		// Prepare Data for writing
		// Repetition ID
		IF (SIf.Cur.dwoJob = RFID_Data.cRFID_AllData) OR (SIf.Cur.dwoJob = RFID_Data.cRFID_RepetionID) THEN
			uinDataAdress := DWORD_TO_UINT(RFID_Data.cRFID_RepetionID);
			uinDataAdress := uinDataAdress MOD 16#100;							// Maximum 255 data
			SIf.Cur.abytData[uinDataAdress] := SIf.Cur.stData.usiRepetitionID;
		END_IF
		// Tray Info
		IF (SIf.Cur.dwoJob = RFID_Data.cRFID_AllData) OR (SIf.Cur.dwoJob = RFID_Data.cRFID_TrayInfo) THEN
			uinDataAdress := DWORD_TO_UINT(RFID_Data.cRFID_TrayInfo);
			uinDataAdress := uinDataAdress MOD 16#100;							// Maximum 255 data
			SIf.Cur.abytData[uinDataAdress].0 := SIf.Cur.stData.bolWorkstation2;
			SIf.Cur.abytData[uinDataAdress].6 := SIf.Cur.stData.bolDeleteFileAfterPrint;
			SIf.Cur.abytData[uinDataAdress].7 := SIf.Cur.stData.bolPrintOk;
		END_IF
		// Height of tray
		IF (SIf.Cur.dwoJob = RFID_Data.cRFID_AllData) OR (SIf.Cur.dwoJob = RFID_Data.cRFID_HeighOfTray) THEN
			uinDataAdress := DWORD_TO_UINT(RFID_Data.cRFID_HeighOfTray);
			uinDataAdress := uinDataAdress MOD 16#100;							// Maximum 255 data
			SIf.Cur.abytData[uinDataAdress] := SHL(SIf.Cur.stData.usiHeightOffset,1);
			SIf.Cur.abytData[uinDataAdress].0 := SIf.Cur.stData.bolHeightUseMeasure;
			SIf.Cur.abytData[uinDataAdress].4 := SIf.Cur.stData.bolHeightOffsetSignMinus;
		END_IF
		// Pretreatment
		IF (SIf.Cur.dwoJob = RFID_Data.cRFID_AllData) OR (SIf.Cur.dwoJob = RFID_Data.cRFID_Pretreatment) THEN
			uinDataAdress := DWORD_TO_UINT(RFID_Data.cRFID_Pretreatment);
			uinDataAdress := uinDataAdress MOD 16#100;							// Maximum 255 data
			SIf.Cur.abytData[uinDataAdress] := SHL(SIf.Cur.stData.usiPlasmaLevel,2);
			SIf.Cur.abytData[uinDataAdress].1 := SIf.Cur.stData.bolIonizer;
			SIf.Cur.abytData[uinDataAdress].4 := SIf.Cur.stData.bolPrintPass;
			SIf.Cur.abytData[uinDataAdress].5 := SIf.Cur.stData.bolNozzleCheck;
			SIf.Cur.abytData[uinDataAdress].6 := SIf.Cur.stData.bolAligneCheck;
		END_IF
		// UV-curing
		IF (SIf.Cur.dwoJob = RFID_Data.cRFID_AllData) OR (SIf.Cur.dwoJob = RFID_Data.cRFID_UVcuring) THEN
			uinDataAdress := DWORD_TO_UINT(RFID_Data.cRFID_UVcuring);
			uinDataAdress := uinDataAdress MOD 16#100;							// Maximum 255 data
			SIf.Cur.abytData[uinDataAdress] := SHL(SIf.Cur.stData.usiUVLampLevel,4);
			IF SIf.Cur.stData.usiUVPinningLevel < 16 THEN // Only 4 bit possible
				usiTemp := SIf.Cur.stData.usiUVPinningLevel OR SIf.Cur.abytData[uinDataAdress];
				SIf.Cur.abytData[uinDataAdress] := usiTemp;
			END_IF
		END_IF
		// Filename
		IF (SIf.Cur.dwoJob = RFID_Data.cRFID_AllData) OR (SIf.Cur.dwoJob = RFID_Data.cRFID_Filename) THEN
			uinDataAdress := DWORD_TO_UINT(RFID_Data.cRFID_Filename);
			uinDataAdress := uinDataAdress MOD 16#100;							// Maximum 255 data
			strTemp := SIf.Cur.stData.strFileName;
			intPositionPoint := TC2_STANDARD.FIND(strTemp,'.');
			IF intPositionPoint > 1 THEN
				intValue := intPositionPoint - 1;
				strTemp := TC2_STANDARD.LEFT(strTemp, intValue);
			END_IF
			intPositionSign := TC2_STANDARD.FIND(strTemp,'-');
			IF intPositionSign > 0 THEN
				intValue :=  TC2_STANDARD.LEN(strTemp) - intPositionSign;
				IF intValue >= 1 THEN
					strTemp := TC2_STANDARD.RIGHT(strTemp, intValue);
					intValue := STRING_TO_INT(strTemp);
					SIf.Cur.abytData[uinDataAdress] := INT_TO_USINT(intValue);
				END_IF
				uliTemp := STRING_TO_ULINT(TC2_STANDARD.LEFT(SIf.Cur.stData.strFileName, (intPositionSign - 1)));
				uinDataLengh := DWORD_TO_UINT(SHR(RFID_Data.cRFID_Filename,16));
				FOR uinTemp := 1 TO  uinDataLengh DO
					SIf.Cur.abytData[uinDataAdress+uinTemp] := ULINT_TO_USINT(uliTemp);
					uliTemp := SHR(uliTemp,8);
				END_FOR
			
			END_IF
		END_IF
				
		// Brush
		IF (SIf.Cur.dwoJob = RFID_Data.cRFID_AllData) OR (SIf.Cur.dwoJob = RFID_Data.cRFID_Brush) THEN
			uinDataAdress := DWORD_TO_UINT(RFID_Data.cRFID_Brush);
			uinDataAdress := uinDataAdress MOD 16#100;							// Maximum 255 data
			SIf.Cur.abytData[uinDataAdress].0 := SIf.Cur.stData.bolBrush;
			SIf.Cur.abytData[uinDataAdress].1 := SIf.Cur.stData.bolBrushClean;
			SIf.Cur.abytData[uinDataAdress].2 := SIf.Cur.stData.bolBrushFans;
			SIf.Cur.abytData[uinDataAdress].6 := SIf.Cur.stData.bolGutterClean;
			SIf.Cur.abytData[uinDataAdress].7 := SIf.Cur.stData.bolSpecialTray;
		END_IF
		
		// Tray ID - not overwritten with all data - fixed name/ID the others are changeable process data
		IF (SIf.Cur.dwoJob = RFID_Data.cRFID_TrayID) THEN	
			uinDataAdress := DWORD_TO_UINT(RFID_Data.cRFID_TrayID);
			uinDataAdress := uinDataAdress MOD 16#100;							// Maximum 255 data
			uinDataLengh := DWORD_TO_UINT(SHR(RFID_Data.cRFID_TrayID,16));
	
			MEMCPY(destAddr:=ADR(SIf.Cur.abytData[uinDataAdress]), srcAddr:=ADR(SIf.Cur.stData.strTrayID), n:=uinDataLengh);
		END_IF
		
		// Write commando
		uinDataAdress := DWORD_TO_UINT(SIf.Cur.dwoJob);
		uinDataAdress := uinDataAdress MOD 16#100;							// Maximum 255 data
		pRFD_SIf^.stCur.uinAdressData := uinDataAdress;
		pRFD_SIf^.stCur.uinAdressTag := DWORD_TO_UINT(SIf.Cur.dwoJob);
		pRFD_SIf^.stCur.usiCount := DWORD_TO_USINT(SHR(SIf.Cur.dwoJob,16));

		IF (CIf.SwCfg.bolSimulation = FALSE) THEN
			pRFD_SIf^.intCmd := RFD_Cmd.cRFD_CMD_Write;
		END_IF
		
	END_IF


//--------------------------------------------------------------------------------------
// Cyclic action
	IF (me.StateMachine.intState=me.StateMachine.intStateLastCycle) THEN

		// Simulation
		IF (CIf.SwCfg.bolSimulation) THEN
			fbSimulationTimer(); // simulation time
			IF (fbSimulationTimer.Q) THEN
				pRFD_SIf^.intCmd := RFD_Cmd.cRFD_CMD_DONE;
			END_IF
		END_IF
		
		//no change action
		 
		
		// State Change Condition
		IF (pRFD_SIf^.stErr.bolErrorActive = TRUE) THEN //  
			me.StateMachine.intStateNext :=  cSTA_ERROR;
		ELSIF (me.StateMachine.udiTimeInState_ms > SIf.Par.udiWriteTime_ms) THEN
			// SIf.Alm[4].strText := 'timeout wait on Data';
			pfbAlarmCtrl^.setAlarm(CIf.Info.intCtrlId,4,0,ADR(SIf.Alm),E_AlmState.RST,CIf.Job.eMe_ActivAlmClass);
			me.StateMachine.intStateNext :=  cSTA_ERROR;
		ELSIF (pRFD_SIf^.intCmd = RFD_Cmd.cRFD_CMD_DONE) THEN
			me.StateMachine.intStateNext := cSTA_WRITE;
		END_IF
	END_IF




//--------------------------------------------------------------------------------------
// Exit action
	IF (me.StateMachine.intState<>me.StateMachine.intStateNext) THEN
		;
	END_IF
END_METHOD

METHOD PROTECTED StateMachine : BOOL
SUPER^.StateMachine();

// main statemachine of base controller
CASE me.StateMachine.intState OF
    RFW_CmdState.cSTA_READBusy: 
        THIS^.sta_READBusy();
    RFW_CmdState.cSTA_READ: 
        THIS^.sta_READ();
    RFW_CmdState.cSTA_WRITEBusy: 
        THIS^.sta_WRITEBusy();
    RFW_CmdState.cSTA_WRITE: 
        THIS^.sta_WRITE();
    RFW_CmdState.cSTA_ONBusy: 
        THIS^.sta_ONBusy();
    RFW_CmdState.cSTA_ON: 
        THIS^.sta_ON();		
    cSTA_RUNBusy: 
        THIS^.sta_RUNBusy();
    cSTA_RUN: 
        THIS^.sta_RUN();		
END_CASE;
END_METHOD

END_FUNCTION_BLOCK

// POUs/Controller/Lvl0/RFW (RFID Reader-Writer)/FB_ULINT_TO_HEXSTRING
FUNCTION FB_ULINT_TO_HEXSTRING : STRING(16)
VAR_INPUT
	in_uliValue: ULINT;
END_VAR
VAR
	intI: INT;
	uliValue: ULINT;
	usiSign: USINT;
	strTemp: STRING(16);
	strSign: STRING(1);
END_VAR

strTemp := '';


	uliValue := in_uliValue;
	
	FOR intI := 0 TO 15 DO
		
		usiSign := ULINT_TO_USINT(uliValue MOD 16);
		uliValue := uliValue/16;
		
		IF usiSign <= 9 THEN		
			strSign := USINT_TO_STRING(usiSign);		// ASCII Sign for Value 16#30 ...16#39
		ELSIF (usiSign = 10) THEN	
			strSign := 'A';
		ELSIF (usiSign = 11) THEN	
			strSign := 'B';
		ELSIF (usiSign = 12) THEN	
			strSign := 'C';
		ELSIF (usiSign = 13) THEN	
			strSign := 'D';
		ELSIF (usiSign = 14) THEN	
			strSign := 'E';
		ELSIF (usiSign = 15) THEN	
			strSign := 'F';
		ELSE
			FB_ULINT_TO_HEXSTRING := '';
			RETURN;
		END_IF
		strTemp := TC2_STANDARD.CONCAT(STR1 := strSign, STR2 := strTemp);
	END_FOR

	FB_ULINT_TO_HEXSTRING := strTemp;

END_FUNCTION

// POUs/Controller/Lvl0/SGT (Signal Tower)/FB_SGT
FUNCTION_BLOCK FB_SGT EXTENDS FB_CtrlBase
VAR_INPUT
	/// Green lamp ON
	In_bolGreenOn: BOOL;
	/// Yellow lamp ON
	In_bolYellowOn: BOOL;
	/// Red lamp ON
	In_bolRedOn: BOOL;
	/// Beep ON
	In_bolBeepOn: BOOL;
	/// Green lamp BLINK
	In_bolGreenBlink: BOOL;
	/// Yellow lamp BLINK
	In_bolYellowBlink: BOOL;
	/// Red lamp BLINK
	In_bolRedBlink: BOOL;
	/// Counter Green (Blink by change, On by Value > 0)
	In_uinCntGreen: UINT;
	/// Counter Yellow (Blink by change, On by Value > 0)
	In_uinCntYellow: UINT;
	/// Counter Red (Blink by change, On by Value > 0)
	In_uinCntRed: UINT;
	/// Counter Beep	(Blink by change, On by Value > 0)
	In_uinCntBeep: UINT;
END_VAR
VAR_OUTPUT
	Out_bolGreen: BOOL;
	Out_bolYellow: BOOL;
	Out_bolRed: BOOL;
	Out_bolBeep: BOOL;
END_VAR
VAR
	/// Shadow copy of In Green Cnt
	uin_InCntGreenOld: UINT;
	/// Shadow copy of In Yellow Cnt
	uin_InCntYellowOld: UINT;
	/// Shadow copy of In Red Cnt
	uin_InCntRedOld: UINT;
	/// Shadow copy of In Beep Cnt
	uin_InCntBeepOld: UINT;
	/// Timer for Oszilator
	udiTimer: UDINT;
	/// Oszilator Signal
	bolTimer: BOOL;
	/// Timer for Beep-Oszilator
	udiBeepTimer: UDINT;
	/// Beep Signal
	bolBeepTimer: BOOL;
	/// Specific interface struct for public access
	SIf: T_Ctrl_SIf_SGT;
END_VAR
VAR CONSTANT
	/// sub States for PONBusy test sequence
	cSTA_SUB_INITIALIZED: INT := 500;
	cSTA_SUB_TestGreen: INT := 502;
	cSTA_SUB_TestYellow: INT := 504;
	cSTA_SUB_TestRed: INT := 506;
	cSTA_SUB_TestBeep: INT := 508;
	cSTA_SUB_FINISH: INT := 510;
END_VAR

(*__________________________________________________________________________________________________
¦	
¦	Vistaprint Schweiz GmbH
¦	CH - 8401 Winterthur
¦
¦	www.vistaprint.ch - info@vistaprint.ch
¦___________________________________________________________________________________________________

Function desription:
Control for the Signal Tower.


History:
Version		Date			Author		Comment
---------------------------------------------------------------------------------------------------
0.00.1		03.06.2014		AVME/MRU	Start history


___________________________________________________________________________________________________*)

SUPER^();

(*
IF (me.bolActivate) THEN // cyclic call enabled
	IF (CIf.Info.bolInitDone=FALSE) THEN // first cycle -> init
		CtrlInit();
		CIf.Info.bolInitDone := TRUE;
	ELSE
		CycleStartDuty();
	
		Always();
		
		StateMachine();
		
		CycleEndDuty();
	END_IF
END_IF;
*)

METHOD PROTECTED Always : BOOL
// not inherite from base !!!
// SUPER^.Always();

IF (me.bolChangeBackToAUTO=TRUE) THEN // switch mode to automatic switch off controller
	//me.StateMachine.intStateNext := cSTA_OFFBusy;
	me.bolChangeBackToAUTO := FALSE; // for cylinder no change to off when switch to automatic!!
END_IF

IF (CIf.SwCfg.bolExist=FALSE) THEN // hardware of controller does not exist
	me.StateMachine.intStateNext := cSTA_SINGLE_ANSWER;
ELSE
	// Init or power on requested -> change to state PONbusy
	IF (((me.StateMachine.intState=cSTA_INITIALIZED) OR (me.intCmd=cCMD_PON)) 
		AND (me.StateMachine.intState<>cSTA_PONBusy) AND (me.StateMachine.intState<>cSTA_PON)
		AND (me.StateMachine.intState<>cSTA_ERROR) AND (me.StateMachine.intState<>cSTA_ERRORQuit) 
		AND (me.StateMachine.intState<>cSTA_EOFF) AND (me.StateMachine.intState<>cSTA_EOFFBusy)) THEN // switch after startup to PONBusy
		me.StateMachine.intStateNext := cSTA_PONBusy;
	END_IF
END_IF

// ----------------------------------------------------------------------------------
// cyclic actions outside of statemachine
IF (me.StateMachine.intState<>cSTA_SINGLE_ANSWER) THEN
	;
END_IF
END_METHOD

PROPERTY PUBLIC CtrlSIf : POINTER TO T_Ctrl_SIf_SGT
GET
END_GET
END_PROPERTY

METHOD FB_init : BOOL
VAR_INPUT
	///if TRUE, the retain variables are initialized (warm start / cold start)
	bInitRetains: BOOL;
	///if TRUE, the instance afterwards gets moved into the copy code (online change)
	bInCopyCode: BOOL;
END_VAR
VAR
	ii: UINT;
END_VAR
//------------------------------------------------------------------------------------------------------------------------
// to manually change in new FUB implementation!!!
// define valid commands for this controller
FOR ii:= 0 TO (SIZEOF(CIf.Job.aCmdList)/SIZEOF(CIf.Job.aCmdList[0])-1) BY 1 DO
	IF (CIf.Job.aCmdList[ii].intCmd=cCMD_INITIALIZED) THEN
		// found first empty array element
		EXIT;
	END_IF
END_FOR

// set name of class/typ
CIf.Info.strType := 'FB_SGT';
CIf.Info.strFullName := 'Signal Tower';

// set alarm class
SIf.Alm[E_ALM_SGT.Dummy].eAlmClass := E_AlmClass.INFO;
SIf.Alm[E_ALM_SGT.Dummy].strText := 'DUMMY';

//*******************************************************************************
// initial values
//*******************************************************************************

// Configuration defaults of class
CIf.SwCfg.bolExist := TRUE;
CIf.SwCfg.bolEnable := TRUE;
CIf.SwCfg.bolSimulation := FALSE;
SIf.Cfg.bolEnableLampTest := TRUE;

// Parameter defaults of class
SIf.Par.udiBlinkTime_ms := 1000;
SIf.Par.udiBeepOnTime_ms := 250;	
SIf.Par.udiBeepOffTime_ms := 2000;
SIf.Par.udiLampTestTime_ms := 500;
END_METHOD

METHOD PROTECTED getCmdState : STRING
VAR_INPUT
	intCmdState: INT;
	bolState: BOOL;
END_VAR
getCmdState := SUPER^.getCmdState(intCmdState:=intCmdState,bolState:=bolState); // get global/base defined cmds/states

IF (getCmdState='') THEN // global not defined get local
	// get string cmd/state string information in runtime
	IF (bolState=FALSE) THEN
		// States's
		CASE intCmdState OF
			(*cCMD_Standby: 
				getCmdState := 'cCMD_Standby'; *)
		END_CASE;  
	ELSE
		// States's
		CASE intCmdState OF
			cSTA_SUB_INITIALIZED: 
				getCmdState := 'cSTA_SUB_INITIALIZED';
			cSTA_SUB_TestGreen: 
				getCmdState := 'cSTA_SUB_TestGreen';
			cSTA_SUB_TestYellow: 
				getCmdState := 'cSTA_SUB_TestYellow';
			cSTA_SUB_TestRed: 
				getCmdState := 'cSTA_SUB_TestRed';
			cSTA_SUB_TestBeep: 
				getCmdState := 'cSTA_SUB_TestBeep';	
			cSTA_SUB_FINISH: 
				getCmdState := 'cSTA_SUB_FINISH';			
		END_CASE;
	END_IF
END_IF
END_METHOD

METHOD getCtrlSIf : POINTER TO T_Ctrl_SIf_SGT
getCtrlSIf := ADR(SIf);
END_METHOD

METHOD PROTECTED IoOutBridge : BOOL
VAR
	bolSwitchValvesOff: BOOL;
END_VAR
// digitale and analoge inputs read from hardware or forcing
IF (CIf.SwCfg.bolSimulation = FALSE) THEN
	setOutBol(CIf.Job.bolIoForce ,ADR(SIf.Out.bolGreen));
	setOutBol(CIf.Job.bolIoForce ,ADR(SIf.Out.bolRed));
	setOutBol(CIf.Job.bolIoForce ,ADR(SIf.Out.bolYellow));
	setOutBol(CIf.Job.bolIoForce ,ADR(SIf.Out.bolBeep));
	
	THIS^.Out_bolGreen := SIf.Out.bolGreen.map;
	THIS^.Out_bolRed := SIf.Out.bolRed.map;
	THIS^.Out_bolYellow := SIf.Out.bolYellow.map;
	THIS^.Out_bolBeep := SIf.Out.bolBeep.map;
END_IF
END_METHOD

METHOD setBeepOutput : BOOL
VAR_INPUT
	/// Oscillate On Input
	bolOscillate: BOOL;
	/// Counter Input
	uinCnt: UINT;
	/// Shadow copy of counter
	uinCntOLD: UINT;
	/// Oscillator Toggle Bit
	bolOscillator: BOOL;
END_VAR
VAR
	bolOscillatorOn: BOOL;
END_VAR
// Beep Oscillate
IF ((uinCnt > uinCntOLD) OR bolOscillate) THEN
	bolOscillatorOn:= TRUE;
END_IF
// Set/Reset Output
IF bolOscillatorOn THEN
	setBeepOutput:= bolOscillator;
ELSE
	setBeepOutput:= FALSE;
END_IF
END_METHOD

METHOD setLampOutput : BOOL
VAR_INPUT
	/// Blink On Input
	bolBlink: BOOL;
	/// Lamp On Input
	bolOn: BOOL;
	/// Counter Input
	uinCnt: UINT;
	/// Shadow copy of counter
	uinCntOLD: UINT;
	/// Oscillator Toggle Bit
	bolOscillator: BOOL;
END_VAR
VAR
	bolBlinkOn: BOOL;
	bolLampOn: BOOL;
END_VAR
// Lamp blink
IF ((uinCnt > uinCntOLD) OR bolBlink) THEN
	bolBlinkOn:= TRUE;
END_IF
// Lamp On
IF ((uinCnt > 0) OR bolOn) THEN
	bolLampOn:= TRUE;
END_IF

// Set/Reset Output
IF bolBlinkOn THEN	// first prio blink
	setLampOutput:= bolOscillator;
ELSIF bolLampOn THEN // second prio 
	setLampOutput:= TRUE;
ELSE
	setLampOutput:= FALSE;
END_IF
END_METHOD

METHOD PROTECTED sta_OFF : BOOL
// state implemetation
//--------------------------------------------------------------------------------------
// Entry action
	IF (me.StateMachine.intState<>me.StateMachine.intStateLastCycle) THEN
		me.StateMachine.intStateLastCycle := me.StateMachine.intState;
		
	END_IF


//--------------------------------------------------------------------------------------
// Cyclic action
	IF (me.StateMachine.intState=me.StateMachine.intStateLastCycle) THEN
		
		;
		
		// State Change Condition
		IF (me.Alarm.eActivAlmClass<>E_AlmClass.EOFF) AND (me.Alarm.eActivAlmClass<>E_AlmClass.OFF) THEN
			IF (me.intCmd=cCMD_RUN) THEN
				me.StateMachine.intStateNext :=  cSTA_RUNBusy;
			END_IF
		END_IF
	END_IF




//--------------------------------------------------------------------------------------
// Exit action
	IF (me.StateMachine.intState<>me.StateMachine.intStateNext) THEN
		;
	END_IF
END_METHOD

METHOD PROTECTED sta_OFFBusy : BOOL
// state implemetation
//--------------------------------------------------------------------------------------
// Entry action
	IF (me.StateMachine.intState<>me.StateMachine.intStateLastCycle) THEN
		me.StateMachine.intStateLastCycle := me.StateMachine.intState;
		// Green Lamp
		SIf.Out.bolGreen.intern := FALSE;
		// Yellow Lamp
		SIf.Out.bolYellow.intern := FALSE;
		// Red Lamp
		SIf.Out.bolRed.intern := FALSE;
		// Beep
		SIf.Out.bolBeep.intern :=FALSE;		
	END_IF

//--------------------------------------------------------------------------------------
// Cyclic action
	IF (me.StateMachine.intState=me.StateMachine.intStateLastCycle) THEN
		
		// State Change Condition
		IF (TRUE) THEN
			me.StateMachine.intStateNext := cSTA_OFF;
		END_IF
	END_IF

//--------------------------------------------------------------------------------------
// Exit action
	IF (me.StateMachine.intState<>me.StateMachine.intStateNext) THEN
		;
	END_IF
END_METHOD

METHOD PROTECTED sta_PON : BOOL
// state implemetation
//--------------------------------------------------------------------------------------
// Entry action
	IF (me.StateMachine.intState<>me.StateMachine.intStateLastCycle) THEN
		me.StateMachine.intStateLastCycle := me.StateMachine.intState;
		
	END_IF


//--------------------------------------------------------------------------------------
// Cyclic action
	IF (me.StateMachine.intState=me.StateMachine.intStateLastCycle) THEN
		
		;
		
		// State Change Condition
		IF(TRUE) THEN // Auto start of Signal Tower
			me.StateMachine.intStateNext := cSTA_RUNBusy;
		END_IF
	END_IF

//--------------------------------------------------------------------------------------
// Exit action
	IF (me.StateMachine.intState<>me.StateMachine.intStateNext) THEN
		;
	END_IF
END_METHOD

METHOD PROTECTED sta_PONBusy : BOOL
// state implemetation
//--------------------------------------------------------------------------------------
// Entry action
	IF (me.StateMachine.intState<>me.StateMachine.intStateLastCycle) THEN
		me.StateMachine.intStateLastCycle := me.StateMachine.intState;
		
		// Green Lamp
		SIf.Out.bolGreen.intern := FALSE;
		// Yellow Lamp
		SIf.Out.bolYellow.intern := FALSE;
		// Red Lamp
		SIf.Out.bolRed.intern := FALSE;
		// Beep
		SIf.Out.bolBeep.intern :=FALSE;	
		
		// Initialize sub state machine
		me.SubStateMachine.intState:= cSTA_SUB_INITIALIZED; 
		me.SubStateMachine.intStateNext:= cSTA_SUB_INITIALIZED;		
	END_IF


//--------------------------------------------------------------------------------------
// Cyclic action
	IF (me.StateMachine.intState=me.StateMachine.intStateLastCycle) THEN

		IF (SIf.Cfg.bolEnableLampTest) THEN
			//--------------------------------------------------------------------------------------
			// sub state machine for lamp test sequence
			CASE me.SubStateMachine.intState OF
				cSTA_SUB_INITIALIZED:
					me.SubStateMachine.intStateNext := cSTA_SUB_TestGreen;
				cSTA_SUB_TestGreen:
					SIf.Out.bolGreen.intern := TRUE;
					IF (me.SubStateMachine.udiTimeInState_ms > SIf.Par.udiLampTestTime_ms) THEN 
						me.SubStateMachine.intStateNext := cSTA_SUB_TestYellow;
					END_IF
				cSTA_SUB_TestYellow:
					SIf.Out.bolYellow.intern := TRUE;
					IF (me.SubStateMachine.udiTimeInState_ms > SIf.Par.udiLampTestTime_ms) THEN 
						me.SubStateMachine.intStateNext := cSTA_SUB_TestRed;
					END_IF			
				cSTA_SUB_TestRed:
					SIf.Out.bolRed.intern := TRUE;
					IF (me.SubStateMachine.udiTimeInState_ms > SIf.Par.udiLampTestTime_ms) THEN 
						me.SubStateMachine.intStateNext := cSTA_SUB_TestBeep;
					END_IF				
				cSTA_SUB_TestBeep:
					SIf.Out.bolBeep.intern := TRUE;
					IF (me.SubStateMachine.udiTimeInState_ms > SIf.Par.udiLampTestTime_ms) THEN
						SIf.Out.bolGreen.intern := FALSE;
						SIf.Out.bolYellow.intern := FALSE;
						SIf.Out.bolRed.intern := FALSE;
						SIf.Out.bolBeep.intern := FALSE; 
						me.SubStateMachine.intStateNext := cSTA_SUB_FINISH;
					END_IF				
				cSTA_SUB_FINISH:
					;
				
			END_CASE
		ELSE // Lamp test not enabled, PONBusy is done
			me.SubStateMachine.intStateNext := cSTA_SUB_FINISH;
		END_IF

		
		// State Change Condition
		IF (me.SubStateMachine.intState = cSTA_SUB_FINISH) THEN	// Test done
			me.StateMachine.intStateNext :=  cSTA_PON;
		END_IF
	END_IF




//--------------------------------------------------------------------------------------
// Exit action
	IF (me.StateMachine.intState<>me.StateMachine.intStateNext) THEN
		;
	END_IF
END_METHOD

METHOD PROTECTED sta_RUN : BOOL
// state implemetation
//--------------------------------------------------------------------------------------
// Entry action
	IF (me.StateMachine.intState<>me.StateMachine.intStateLastCycle) THEN
		me.StateMachine.intStateLastCycle := me.StateMachine.intState;

	END_IF


//--------------------------------------------------------------------------------------
// Cyclic action
	IF (me.StateMachine.intState=me.StateMachine.intStateLastCycle) THEN

		// Simulation
		IF (CIf.SwCfg.bolSimulation) THEN
			;
		END_IF
		
		// Oscillator for blinking lamp
		IF (udiTimer >= 2*SIf.Par.udiBlinkTime_ms) THEN
			bolTimer:= FALSE;
			udiTimer:= 0;
		ELSIF (udiTimer >= SIf.Par.udiBlinkTime_ms) THEN
			bolTimer:= TRUE;
		END_IF
		udiTimer:= udiTimer + me.FUBInfo.udiSample_ms;
		// Oscillator for Beep
		IF (udiBeepTimer >= (SIf.Par.udiBeepOffTime_ms + SIf.Par.udiBeepOnTime_ms)) THEN
			bolBeepTimer:= TRUE;
			udiBeepTimer:= 0;
		ELSIF (udiBeepTimer >= SIf.Par.udiBeepOnTime_ms) THEN
			bolBeepTimer:= FALSE;
		END_IF
		udiBeepTimer:= udiBeepTimer + me.FUBInfo.udiSample_ms;	
		
		// Green Lamp
		SIf.Out.bolGreen.intern := setLampOutput(bolBlink:= In_bolGreenBlink, bolOn:= In_bolGreenOn, uinCnt:= In_uinCntGreen, 
												uinCntOLD:= uin_InCntGreenOld, bolOscillator:= bolTimer);
		// Yellow Lamp
		SIf.Out.bolYellow.intern := setLampOutput(bolBlink:= In_bolYellowBlink, bolOn:= In_bolYellowOn, uinCnt:= In_uinCntYellow, 
												uinCntOLD:= uin_InCntYellowOld, bolOscillator:= bolTimer);
		// Red Lamp
		SIf.Out.bolRed.intern := setLampOutput(bolBlink:= In_bolRedBlink, bolOn:= In_bolRedOn, uinCnt:= In_uinCntRed, 
												uinCntOLD:= uin_InCntRedOld, bolOscillator:= bolTimer);
		// Beep										
		SIf.Out.bolBeep.intern := setBeepOutput(bolOscillate:= In_bolBeepOn, uinCnt:= In_uinCntBeep,
												uinCntOLD:= uin_InCntBeepOld, bolOscillator:= bolBeepTimer);
												
		// Reset
		IF (CIf.Job.bolAlmReset) THEN
			uin_InCntGreenOld:= In_uinCntGreen;
			uin_InCntYellowOld:= In_uinCntYellow;
			uin_InCntRedOld:= In_uinCntRed;
			uin_InCntBeepOld:= In_uinCntBeep;
			CIf.Job.bolAlmReset := FALSE;
		END_IF
		
		// State Change Condition
		IF(me.intCmd=cCMD_OFF) THEN
			me.StateMachine.intStateNext := cSTA_OFFBusy;
		END_IF
	END_IF



//--------------------------------------------------------------------------------------
// Exit action
	IF (me.StateMachine.intState<>me.StateMachine.intStateNext) THEN
		;
	END_IF
END_METHOD

METHOD PROTECTED sta_RUNBusy : BOOL
// state implemetation
//--------------------------------------------------------------------------------------
// Entry action
	IF (me.StateMachine.intState<>me.StateMachine.intStateLastCycle) THEN
		me.StateMachine.intStateLastCycle := me.StateMachine.intState;

	END_IF


//--------------------------------------------------------------------------------------
// Cyclic action
	IF (me.StateMachine.intState=me.StateMachine.intStateLastCycle) THEN

		
		// State Change Condition
		IF (TRUE) THEN
			me.StateMachine.intStateNext := cSTA_RUN;
		END_IF
	END_IF


//--------------------------------------------------------------------------------------
// Exit action
	IF (me.StateMachine.intState<>me.StateMachine.intStateNext) THEN
		;
	END_IF
END_METHOD

METHOD PROTECTED StateMachine : BOOL
SUPER^.StateMachine();

// main statemachine of base controller
CASE me.StateMachine.intState OF
	cSTA_RUN:
		THIS^.sta_RUN();
	cSTA_RUNBusy:
		THIS^.sta_RUNBusy();
END_CASE;
END_METHOD

END_FUNCTION_BLOCK

// POUs/Controller/Lvl0/UMC [Universal Motor Controller]/FB_UMC
FUNCTION_BLOCK FB_UMC EXTENDS FB_CtrlBase
VAR_INPUT
	In_uinStatus				: UINT;
	In_intMotorActualSpeed		: INT;
	In_uinMotorSetSpeed			: UINT;
	In_strNetId					: AMSNETID;
	In_uintPort					: WORD;
	In_uinECATState				: UINT;
	In_bolEmoOk					: BOOL;
END_VAR
VAR_OUTPUT
	Out_uinControl      	: UINT;
	Out_uinSpeedSetpoint	: UINT;
END_VAR
VAR
	/// Specific interface struct for public access
	SIf					: T_Ctrl_SIf_UMC;
	In_unStatus			: U_UMC_Lenze_Status;
	Out_unControl		: U_UMC_Lenze_Control;
	arTurnDirection		: ARRAY[0..MAX_E_TURN_DIRECTION] OF BOOL;
	fbPulse				: TC2_STANDARD.TP;
	/// EtherCAT slave diagnostics via CoE
	fbEcCoESdoRead_ErrorText: FB_EcCoESdoRead;
	sErrorText: STRING(80);
	sNetId: T_AmsNetId;
	bSdoRead: BOOL;
END_VAR
VAR CONSTANT
	cLEFT				: BOOL := TRUE;
	cRIGHT				: BOOL := FALSE;

	cEtherCAT_OP_MODE		: UINT := 16#0008;
	cEtherCAT_MODE_MASK		: UINT := 16#000F;
END_VAR

(*__________________________________________________________________________________________________
¦	
¦	Vistaprint Schweiz GmbH
¦	CH - 8401 Winterthur
¦
¦	www.vistaprint.ch - info@vistaprint.ch
¦___________________________________________________________________________________________________

Function desription:
Lenze Motor implementation. 


History:
Version		Date			Author		Comment
---------------------------------------------------------------------------------------------------
0.00.1		09.07.2013		PC			Start history
0.00.2		04.02.2014		AVM/MRU		Simulation mode
										cCMD_LEFT / cCMD_RIGHT added in FB_init / getCmdState
0.00.3		02.10.2014		AVM/MRU		SingleAnswer in Always added
0.00.4		05.12.2014		HLV/MAH		Motor status information text from CoE added

___________________________________________________________________________________________________*)

SUPER^();

(*
IF (me.bolActivate) THEN // cyclic call enabled
	IF (CIf.Info.bolInitDone=FALSE) THEN // first cycle -> init
		CtrlInit();
		CIf.Info.bolInitDone := TRUE;
	ELSE
		CycleStartDuty();
	
		Always();
		
		StateMachine();
		
		CycleEndDuty();
	END_IF
END_IF;
*)

METHOD PROTECTED Always : BOOL
//SUPER^.Always();

IF (me.bolChangeBackToAUTO=TRUE) THEN // switch mode to automatic switch off controller
	me.StateMachine.intStateNext := cSTA_OFFBusy;
	me.bolChangeBackToAUTO := FALSE;
END_IF

IF (CIf.SwCfg.bolExist=FALSE) THEN // hardware of controller does not exist
	me.StateMachine.intStateNext := cSTA_SINGLE_ANSWER;
ELSE
    IF (((me.StateMachine.intState=cSTA_INITIALIZED) OR (me.intCmd=cCMD_PON)) 
        AND (me.StateMachine.intState<>cSTA_PONBusy) AND (me.StateMachine.intState<>cSTA_PON)
        AND (me.StateMachine.intState<>cSTA_ERROR) AND (me.StateMachine.intState<>cSTA_ERRORQuit) 
        AND (me.StateMachine.intState<>cSTA_EOFF) AND (me.StateMachine.intState<>cSTA_EOFFBusy)) THEN // switch after startup to PONBusy
        me.StateMachine.intStateNext := cSTA_PONBusy;
    END_IF
END_IF

// ----------------------------------------------------------------------------------
// Simulation
IF (CIf.SwCfg.bolSimulation) THEN
	// Simulate inputs (no physical inputs)
	SIf.In.bolEmoOk.intern := TRUE;
END_IF

// ----------------------------------------------------------------------------------
// Conditions Always
IF (me.StateMachine.intState<>cSTA_SINGLE_ANSWER) THEN
	
	IF (((me.StateMachine.intState=cSTA_INITIALIZED) OR (me.intCmd=cCMD_PON))
		AND (me.StateMachine.intState<>cSTA_PONBusy) AND (me.StateMachine.intState<>cSTA_PON)
		AND (me.StateMachine.intState<>cSTA_ERROR) AND (me.StateMachine.intState<>cSTA_ERRORQuit)
		AND (me.StateMachine.intState<>cSTA_EOFF) AND (me.StateMachine.intState<>cSTA_EOFFBusy)) THEN
		me.StateMachine.intStateNext := cSTA_PONBusy;
	END_IF

	IF (((me.Alarm.eActivAlmClass=E_AlmClass.OFF) OR (me.intCmd=cCMD_OFF))
			AND (me.StateMachine.intState<>cSTA_ERROR) AND (me.StateMachine.intState<>cSTA_ERRORQuit)
			AND (me.StateMachine.intState<>cSTA_EOFF) AND (me.StateMachine.intState<>cSTA_EOFFBusy)
			AND (me.StateMachine.intState<>cSTA_OFF) AND (me.StateMachine.intState<>cSTA_OFFBusy)
			AND (me.StateMachine.intState<>UMC_CmdState.cSTA_RESETMOTORERROR) 
			AND (me.StateMachine.intState<>UMC_CmdState.cSTA_SETOPERATIONMODE)) THEN
		me.StateMachine.intStateNext := cSTA_OFFBusy;	
	END_IF

	IF ((SIf.In.bolEmoOk.intern = FALSE) AND (me.StateMachine.intState <> cSTA_EOFF) 
		AND (me.StateMachine.intState <> BASE_PLC.cSTA_EOFFBusy)
		AND (me.StateMachine.intState <> BASE_PLC.cSTA_ERROR) 
		AND (me.StateMachine.intState <> BASE_PLC.cSTA_PON) 
		AND (me.StateMachine.intState <> BASE_PLC.cSTA_PONBusy) 
		AND (me.StateMachine.intState<>BASE_PLC.cSTA_INITIALIZED)
		AND (me.StateMachine.intState <> BASE_PLC.cSTA_ERRORQuit)) THEN
		me.StateMachine.intStateNext := cSTA_EOFFBusy;				
	END_IF
	
END_IF
END_METHOD

METHOD PROTECTED cmd_MotorOff : BOOL
Out_unControl.Output 				:= 0;
Out_unControl.Data.SetDCBreak 		:= 1;
Out_unControl.Data.SetHalt        	:= 1;
Out_unControl.Data.SetQuickStop    	:= 1;
SIf.Out.uinSpeedSetpoint.intern 	:= 0;
END_METHOD

METHOD PROTECTED cmd_MotorOn : BOOL
VAR_INPUT
	bDirection		: BOOL;		// Direction of the drive; False = Right; True = Left
	uinSpeed		: UINT;					// Speed of the belt
END_VAR
Out_unControl.Output 				:= 0;
Out_unControl.Data.EnableOperation 	:= 1;
Out_unControl.Data.SwitchOn        	:= 1;
Out_unControl.Data.SetSpeedCcw     	:= bDirection;

SIf.Out.uinSpeedSetpoint.intern 	:= uinSpeed;
END_METHOD

METHOD PROTECTED cmd_MotorReset : BOOL
VAR_INPUT
END_VAR
cmd_MotorOff();
Out_unControl.Data.ResetFault 		:= 1;
END_METHOD

METHOD PROTECTED cmd_MotorStop : BOOL
VAR_INPUT
END_VAR
Out_unControl.Output 				:= 0;
Out_unControl.Data.SetDCBreak 		:= 1;
Out_unControl.Data.SetHalt        	:= 1;
Out_unControl.Data.SetQuickStop    	:= 1;
END_METHOD

METHOD PUBLIC CtrlInit : BOOL
VAR_INPUT
END_VAR
SUPER^.CtrlInit();

arTurnDirection[E_TURN_DIRECTION.AUTOMATIC] := FALSE;
arTurnDirection[E_TURN_DIRECTION.LEFT] 		:= FALSE;
arTurnDirection[E_TURN_DIRECTION.RIGHT] 	:= TRUE;

SIf.Cur.uinSpeedLimit := SIf.Cfg.uinMaxSpeed * SIf.Cfg.uinLC11_100 / 100;
END_METHOD

PROPERTY PUBLIC CtrlSIf : POINTER TO T_Ctrl_SIf_UMC
GET
CtrlSIf := ADR(SIf);
END_GET
END_PROPERTY

METHOD PROTECTED CycleEndDuty : BOOL
VAR_INPUT
END_VAR
SIf.Out.uinControl.intern := Out_unControl.Output;

SUPER^.CycleEndDuty();
END_METHOD

METHOD PROTECTED CycleStartDuty : BOOL
VAR_INPUT
END_VAR
SUPER^.CycleStartDuty();

In_unStatus.Input := SIf.In.uinStatus.intern;
END_METHOD

METHOD FB_init : BOOL
VAR_INPUT
	bInitRetains : BOOL; // if TRUE, the retain variables are initialized (warm start / cold start)
	bInCopyCode : BOOL;  // if TRUE, the instance afterwards gets moved into the copy code (online change)
END_VAR
VAR
	iIdx		: UINT;
	iLength		: UINT;	
END_VAR
//------------------------------------------------------------------------------------------------------------------------
// to manually change in new FUB implementation!!!
// define valid commands for this controller
iLength := SIZEOF(CIf.Job.aCmdList)/SIZEOF(CIf.Job.aCmdList[0]);
iIdx := 0;

WHILE (iIdx < iLength) AND (CIf.Job.aCmdList[iIdx].intCmd <> cCMD_INITIALIZED) DO
	iIdx := iIdx + 1; 
END_WHILE

IF (iIdx < iLength) THEN
// Add configuration of own comands	
	CIf.Job.aCmdList[iIdx].intCmd := BASE_PLC.cCMD_STOP;
	CIf.Job.aCmdList[iIdx].strName := 'Stop'; 
	CIf.Job.aCmdList[iIdx].bolAvailable := TRUE;
	iIdx := iIdx + 1;
	CIf.Job.aCmdList[iIdx].intCmd := cCMD_RUN;
	CIf.Job.aCmdList[iIdx].strName := 'Run'; 
	CIf.Job.aCmdList[iIdx].bolAvailable := TRUE;
	iIdx := iIdx + 1;
	CIf.Job.aCmdList[iIdx].intCmd := cCMD_LEFT;
	CIf.Job.aCmdList[iIdx].strName := 'Left'; 
	CIf.Job.aCmdList[iIdx].bolAvailable := TRUE;
	iIdx := iIdx + 1;
	CIf.Job.aCmdList[iIdx].intCmd := cCMD_RIGHT;
	CIf.Job.aCmdList[iIdx].strName := 'Right'; 
	CIf.Job.aCmdList[iIdx].bolAvailable := TRUE;
	iIdx := iIdx + 1;
ELSE
	;// Error if the aCmdList Array is to small
END_IF

// set name of class/typ
CIf.Info.strType := 'FB_UMC';
CIf.Info.strFullName := 'Universal Motor Controller';

// set alarm class
SIf.Alm[E_ALM_UMC.MotorOnTimeout].eAlmClass := Base_PLC.E_AlmClass.TSTOP;
SIf.Alm[E_ALM_UMC.MotorOnTimeout].strText := 'Motor On Timeout'; 
SIf.Alm[E_ALM_UMC.MotorError].eAlmClass := Base_PLC.E_AlmClass.TSTOP;
SIf.Alm[E_ALM_UMC.MotorError].strText := 'Motor Error';
SIf.Alm[E_ALM_UMC.MotorWarning].eAlmClass := Base_PLC.E_AlmClass.WARNING;
SIf.Alm[E_ALM_UMC.MotorWarning].strText := 'Motor Warning';
SIf.Alm[E_ALM_UMC.MotorOverCurrent].eAlmClass := Base_PLC.E_AlmClass.WARNING;
SIf.Alm[E_ALM_UMC.MotorOverCurrent].strText := 'Motor Over Current';
SIf.Alm[E_ALM_UMC.MotorNotReady].eAlmClass := Base_PLC.E_AlmClass.TSTOP;
SIf.Alm[E_ALM_UMC.MotorNotReady].strText := 'Motor Not Ready';
SIf.Alm[E_ALM_UMC.DirectionParameterOverflow].eAlmClass := Base_PLC.E_AlmClass.TSTOP;
SIf.Alm[E_ALM_UMC.DirectionParameterOverflow].strText := 'Direction Parameter Overflow';
SIf.Alm[E_ALM_UMC.SpeedOverLimit].eAlmClass := Base_PLC.E_AlmClass.WARNING;
SIf.Alm[E_ALM_UMC.SpeedOverLimit].strText := 'Motor Setpoint over the limit';
SIf.Alm[E_ALM_UMC.MotorStatusInformation].eAlmClass := Base_PLC.E_AlmClass.INFO;

//*******************************************************************************
// initial values
//*******************************************************************************

// software configuration
CIf.SwCfg.bolExist := TRUE;
CIf.SwCfg.bolEnable := TRUE;
CIf.SwCfg.bolSimulation := FALSE;

// configuration
SIf.Cfg.uinLC11 := 1500;
SIf.Cfg.uinLC11_100 := 16384;
SIf.Cfg.uinMaxSpeed := 150;

// parameter
SIf.Par.udiStartupOnTime_ms := 5000;
SIf.Par.udiMotorOnTime_ms 	:= 10000;
SIf.Par.uinSpeed_rpm 		:= 1000;
SIf.Par.uinMotorResetPulseTime_ms	:= 500;
SIf.Par.uinMotorResetCnt 		:= 3;
SIf.Par.udiMoveStartLatency 	:= 15;
SIf.Par.udiMoveStopLatency 		:= 60;
SIf.Par.eRotationDirection  := E_TURN_DIRECTION.LEFT;

SIf.Par.udiSimMotorOnTime_ms := SIf.Par.udiMotorOnTime_ms / 10;
END_METHOD

METHOD PROTECTED getCmdState : STRING

VAR_INPUT
	intCmdState: INT;
	bolState: BOOL;
END_VAR
getCmdState := SUPER^.getCmdState(intCmdState:=intCmdState,bolState:=bolState); // get global/base defined cmds/states

IF (getCmdState='') THEN // global not defined get local
	// get string cmd/state string information in runtime
	IF (bolState=FALSE) THEN
		// Comands's
		CASE intCmdState OF
			cCMD_LEFT: 
				getCmdState := 'cCMD_Left';
			cCMD_RIGHT: 
				getCmdState := 'cCMD_Right';
		END_CASE;
	ELSE
		// States's
		CASE intCmdState OF
			cSTA_RUN: 
				getCmdState := 'RUN';
			cSTA_RUNBusy: 
				getCmdState := 'RUNBusy';
			UMC_CmdState.cSTA_RESETMOTORERROR:
				getCmdState := 'RESETMOTORERROR';
			UMC_CmdState.cSTA_SETOPERATIONMODE:
				getCmdState := 'SETOPERATIONMODE';
		END_CASE;
	END_IF
END_IF
END_METHOD

METHOD getCtrlSIf : POINTER TO T_Ctrl_SIf_UMC
getCtrlSIf := ADR(SIf);
END_METHOD

METHOD PROTECTED GetMotorStatus : E_UMC_MOTOR_STATUS
VAR_INPUT
	uinMotorStatus		: UINT;
END_VAR
uinMotorStatus := uinMotorStatus AND 16#0F00;
uinMotorStatus := SHR(uinMotorStatus,8);
GetMotorStatus := UINT_TO_INT(uinMotorStatus);
END_METHOD

METHOD PROTECTED GetSpeedValue : UINT
VAR
	uinSpeedOutput			: UINT;
END_VAR
uinSpeedOutput := SIf.Par.uinSpeed_rpm * SIf.Cfg.uinLC11_100 / SIf.Cfg.uinLC11;

IF uinSpeedOutput > SIf.Cur.uinSpeedLimit THEN
	uinSpeedOutput := SIf.Cur.uinSpeedLimit;
	pfbAlarmCtrl^.setAlarm(CIf.Info.intCtrlId,INT_TO_UINT(E_ALM_UMC.SpeedOverLimit),0,ADR(SIf.Alm),E_AlmState.RST,CIf.Job.eMe_ActivAlmClass);
END_IF

GetSpeedValue := uinSpeedOutput;
END_METHOD

METHOD PROTECTED IoInBridge : BOOL
// digitale and analoge inputs read from hardware or forcing
SIf.In.uinStatus.map			:= THIS^.In_uinStatus				;
SIf.In.intMotorActualSpeed.map	:= THIS^.In_intMotorActualSpeed	;
SIf.In.uinMotorSetSpeed.map		:= THIS^.In_uinMotorSetSpeed		;
SIf.In.bolEmoOk.map				:= THIS^.In_bolEmoOk		;

IF (CIf.SwCfg.bolSimulation = FALSE) THEN
	BASE_PLC.getInUint(CIf.Job.bolIoForce,ADR(SIf.In.uinStatus));
	BASE_PLC.getInUint(CIf.Job.bolIoForce,ADR(SIf.In.intMotorActualSpeed));
	BASE_PLC.getInUint(CIf.Job.bolIoForce,ADR(SIf.In.uinMotorSetSpeed));
	BASE_PLC.getInUint(CIf.Job.bolIoForce,ADR(SIf.In.bolEmoOk));
ELSE
	//simulation of global IO
END_IF
END_METHOD

METHOD PROTECTED IoOutBridge : BOOL
VAR
	bolSwitchValvesOff: BOOL;
END_VAR
// digitale and analoge inputs read from hardware or forcing
IF (CIf.SwCfg.bolSimulation = FALSE) THEN
	BASE_PLC.setOutUint(CIf.Job.bolIoForce ,ADR(SIf.Out.uinControl));
	BASE_PLC.setOutUint(CIf.Job.bolIoForce ,ADR(SIf.Out.uinSpeedSetpoint));

	THIS^.Out_uinControl			:= SIf.Out.uinControl.map	;
	THIS^.Out_uinSpeedSetpoint		:= SIf.Out.uinSpeedSetpoint.map	;
END_IF
END_METHOD

METHOD PROTECTED sta_EOFF : BOOL
VAR_INPUT
END_VAR
// state implemetation
//--------------------------------------------------------------------------------------
// Entry action
	IF (me.StateMachine.intState<>me.StateMachine.intStateLastCycle) THEN
		me.StateMachine.intStateLastCycle := me.StateMachine.intState;	
	END_IF

//--------------------------------------------------------------------------------------
// Cyclic action
	IF (me.StateMachine.intState=me.StateMachine.intStateLastCycle) THEN		
		// As long as the EMO is not reseted!
		IF SIf.In.bolEmoOk.intern THEN
			IF me.StateMachine.intStateHistory=cSTA_PONBusy OR me.StateMachine.intStateHistory=cSTA_PON THEN
				me.StateMachine.intStateNext := BASE_PLC.cSTA_PONBusy;
			ELSE
				me.StateMachine.intStateNext := BASE_PLC.cSTA_OFFBusy;
			END_IF
		ELSE
			IF me.intCmd <> BASE_PLC.cCMD_OFF THEN
				// Clear pending and new commands cyclic to prevent automatic recovery!	
				CIf.Job.intACmd := BASE_PLC.cCMD_DONE;
				CIf.Job.intMCmd := BASE_PLC.cCMD_DONE;		
			END_IF
		END_IF
	END_IF

//--------------------------------------------------------------------------------------
// Exit action
	IF (me.StateMachine.intState<>me.StateMachine.intStateNext) THEN
		;
	END_IF
END_METHOD

METHOD PROTECTED sta_EOFFbusy : BOOL
VAR_INPUT
END_VAR
// state implemetation
//--------------------------------------------------------------------------------------
// Entry action
IF (me.StateMachine.intState<>me.StateMachine.intStateLastCycle) THEN
	me.StateMachine.intStateHistory := me.StateMachine.intStateLastCycle;
	me.StateMachine.intStateLastCycle := me.StateMachine.intState;
	
	cmd_MotorOff();
END_IF

//--------------------------------------------------------------------------------------
// Cyclic action
IF (me.StateMachine.intState=me.StateMachine.intStateLastCycle) THEN
	IF (TRUE) THEN
		me.StateMachine.intStateNext := BASE_PLC.cSTA_EOFF;
	END_IF
END_IF

//--------------------------------------------------------------------------------------
// Exit action
IF (me.StateMachine.intState<>me.StateMachine.intStateNext) THEN
	;
END_IF
END_METHOD

METHOD PROTECTED sta_ERROR : BOOL
// state implemetation
//--------------------------------------------------------------------------------------
// Entry action
	IF (me.StateMachine.intState<>me.StateMachine.intStateLastCycle) THEN
		me.StateMachine.intStateHistory := me.StateMachine.intStateLastCycle; // -> possibillity to go back to state before error
		me.StateMachine.intStateLastCycle := me.StateMachine.intState;
		SIf.Cur.uinMotorResetCnt := 0;
		cmd_MotorOff();
		
		bSdoRead := TRUE;
	END_IF


//--------------------------------------------------------------------------------------
// Cyclic action
	IF (me.StateMachine.intState=me.StateMachine.intStateLastCycle) THEN
		
		sNetId := F_CreateAmsNetId(In_strNetId);
		fbEcCoESdoRead_ErrorText(sNetId := sNetId,
								 nSlaveAddr := WORD_TO_UINT(In_uintPort),
								 nSubIndex := 3,
								 nIndex := 16#5F59,
								 pDstBuf := ADR(sErrorText),
								 cbBufLen := 70,
								 bExecute := bSdoRead,
								 tTimeout := T#500MS);
								 
		IF bSdoRead AND NOT fbEcCoESdoRead_ErrorText.bBusy THEN
			bSdoRead := FALSE;
		END_IF
		
		IF F_toUCase(sErrorText) <> 'NO ERROR' THEN
			SIf.Alm[E_ALM_UMC.MotorStatusInformation].strText := sErrorText;
			pfbAlarmCtrl^.setAlarm(CIf.Info.intCtrlId,INT_TO_UINT(E_ALM_UMC.MotorStatusInformation),0,ADR(SIf.Alm),E_AlmState.RST,CIf.Job.eMe_ActivAlmClass);
		END_IF
		
		// State Change Condition
		IF (CIf.Job.bolAlmReset = TRUE) THEN
			me.StateMachine.intStateNext := cSTA_ERRORQuit;
		END_IF
	END_IF




//--------------------------------------------------------------------------------------
// Exit action
	IF (me.StateMachine.intState<>me.StateMachine.intStateNext) THEN
		;
	END_IF
END_METHOD

METHOD PROTECTED sta_ERRORQuit : BOOL
// state implemetation
//--------------------------------------------------------------------------------------
// Entry action
	IF (me.StateMachine.intState<>me.StateMachine.intStateLastCycle) THEN
		me.StateMachine.intStateLastCycle := me.StateMachine.intState;
		
	END_IF


//--------------------------------------------------------------------------------------
// Cyclic action
	IF (me.StateMachine.intState=me.StateMachine.intStateLastCycle) THEN
		
		;
		// evtl. wait time if reset of device is necessary and then decide to go to states or ERROR state
		IF (CIf.Job.bolAlmReset = TRUE) THEN
			CIf.Job.eMe_ActivAlmClass := E_AlmClass.NONE; // reset feedback channel for parent
			CIf.Job.bolAlmReset := FALSE;
		END_IF
		
		// State Change Condition
		IF (CIf.Job.bolAlmReset = FALSE) THEN
			IF (me.StateMachine.intStateHistory<=cSTA_PON) THEN
				me.StateMachine.intStateNext := cSTA_PON;
			ELSIF (CIf.SwCfg.bolSimulation = TRUE) THEN	// Do not set operation mode in simulation
				me.StateMachine.intStateNext := BASE_PLC.cSTA_OFF;
			ELSE
				me.StateMachine.intStateNext := UMC_CmdState.cSTA_SETOPERATIONMODE;
			END_IF
		END_IF
	END_IF




//--------------------------------------------------------------------------------------
// Exit action
	IF (me.StateMachine.intState<>me.StateMachine.intStateNext) THEN
		;
	END_IF
END_METHOD

METHOD PROTECTED sta_OFF : BOOL
VAR_INPUT
END_VAR
// state implemetation
//--------------------------------------------------------------------------------------
// Entry action
	IF (me.StateMachine.intState<>me.StateMachine.intStateLastCycle) THEN
		me.StateMachine.intStateLastCycle := me.StateMachine.intState;

		SIf.Cur.uinMotorResetCnt := 0;
	END_IF


//--------------------------------------------------------------------------------------
// Cyclic action
	IF (me.StateMachine.intState=me.StateMachine.intStateLastCycle) THEN
		CASE me.intCmd OF
			cCMD_Left:
				SIf.Par.eRotationDirection := E_TURN_DIRECTION.LEFT;
				me.StateMachine.intStateNext := cSTA_RUNBusy;
			cCMD_Right:
				SIf.Par.eRotationDirection := E_TURN_DIRECTION.RIGHT;
				me.StateMachine.intStateNext := cSTA_RUNBusy;
			BASE_PLC.cCMD_STOP:
				me.StateMachine.intStateNext := BASE_PLC.cSTA_STOPBusy;
			BASE_PLC.cCMD_RUN:
				me.StateMachine.intStateNext := cSTA_RUNBusy;
		END_CASE
	END_IF


//--------------------------------------------------------------------------------------
// Exit action
	IF (me.StateMachine.intState<>me.StateMachine.intStateNext) THEN
		;
	END_IF
END_METHOD

METHOD PROTECTED sta_OFFBusy : BOOL
VAR
	uinECatStatus	: UINT;
	eMotorStatus	: E_UMC_MOTOR_STATUS;
END_VAR
// state implemetation
//--------------------------------------------------------------------------------------
// Entry action
	IF (me.StateMachine.intState<>me.StateMachine.intStateLastCycle) THEN
		me.StateMachine.intStateLastCycle := me.StateMachine.intState;
		cmd_MotorOff();
	END_IF


//--------------------------------------------------------------------------------------
// Cyclic action
	IF (me.StateMachine.intState=me.StateMachine.intStateLastCycle) THEN
		eMotorStatus := GetMotorStatus(sif.In.uinStatus.intern);
		uinECatStatus := In_uinECATState AND cEtherCAT_MODE_MASK;

		IF    (uinECatStatus = cEtherCAT_OP_MODE)
		  AND NOT In_unStatus.Data.Trouble 
		  AND In_unStatus.Data.ActSpeedIsZero
		  AND (eMotorStatus = E_UMC_MOTOR_STATUS.ReadyToSwitchON) THEN
			me.StateMachine.intStateNext := Base_PLC.cSTA_OFF;
		ELSIF (CIf.SwCfg.bolSimulation = TRUE) THEN	// Do not set operation mode in simulation
			me.StateMachine.intStateNext := BASE_PLC.cSTA_OFF;
		ELSE
			IF me.StateMachine.udiTimeInState_ms > SIf.Par.uinMotorResetPulseTime_ms THEN
				IF SIf.Cur.uinMotorResetCnt > SIf.Par.uinMotorResetCnt THEN
					pfbAlarmCtrl^.setAlarm(CIf.Info.intCtrlId,INT_TO_UINT(E_ALM_UMC.MotorError),0,ADR(SIf.Alm),E_AlmState.RST,CIf.Job.eMe_ActivAlmClass);
					me.StateMachine.intStateNext := Base_PLC.cSTA_ERROR;	
				ELSE
					me.StateMachine.intStateNext := UMC_CmdState.cSTA_SETOPERATIONMODE;
				END_IF
			END_IF
		END_IF
	END_IF

//--------------------------------------------------------------------------------------
// Exit action
	IF (me.StateMachine.intState<>me.StateMachine.intStateNext) THEN
		;
	END_IF
END_METHOD

METHOD PROTECTED sta_PON : BOOL
VAR_INPUT
END_VAR
// state implemetation
//--------------------------------------------------------------------------------------
// Entry action
	IF (me.StateMachine.intState<>me.StateMachine.intStateLastCycle) THEN
		me.StateMachine.intStateLastCycle := me.StateMachine.intState;
	END_IF


//--------------------------------------------------------------------------------------
// Cyclic action
	IF (me.StateMachine.intState=me.StateMachine.intStateLastCycle) THEN
		;
	END_IF


//--------------------------------------------------------------------------------------
// Exit action
	IF (me.StateMachine.intState<>me.StateMachine.intStateNext) THEN
		;
	END_IF
END_METHOD

METHOD PROTECTED sta_RESETMOTORERROR : BOOL
VAR
	eMotorStatus	: E_UMC_MOTOR_STATUS;
END_VAR
// state implemetation
//--------------------------------------------------------------------------------------
// Entry action
	IF (me.StateMachine.intState<>me.StateMachine.intStateLastCycle) THEN
		me.StateMachine.intStateLastCycle := me.StateMachine.intState;
		cmd_MotorReset();
	END_IF


//--------------------------------------------------------------------------------------
// Cyclic action
	IF (me.StateMachine.intState=me.StateMachine.intStateLastCycle) THEN
		eMotorStatus := GetMotorStatus(sif.In.uinStatus.intern);

		IF me.SubStateMachine.udiTimeInState_ms > SIf.Par.uinMotorResetPulseTime_ms THEN
			SIf.Cur.uinMotorResetCnt := SIf.Cur.uinMotorResetCnt + 1;
			me.StateMachine.intStateNext := BASE_PLC.cSTA_OFFBusy;
		END_IF
	END_IF


//--------------------------------------------------------------------------------------
// Exit action
	IF (me.StateMachine.intState<>me.StateMachine.intStateNext) THEN
		Out_unControl.Data.ResetFault := FALSE;
	END_IF
END_METHOD

METHOD PROTECTED sta_RUN : BOOL
VAR
	uniStatus 		: U_UMC_Lenze_Status;
END_VAR
// state implemetation
//--------------------------------------------------------------------------------------
// Entry action
	IF (me.StateMachine.intState<>me.StateMachine.intStateLastCycle) THEN
		me.StateMachine.intStateLastCycle := me.StateMachine.intState;
		CIf.Job.intACmd := BASE_PLC.cCMD_DONE;
	END_IF


//--------------------------------------------------------------------------------------
// Cyclic action
	IF (me.StateMachine.intState=me.StateMachine.intStateLastCycle) THEN
		IF In_unStatus.Data.Trouble THEN
			pfbAlarmCtrl^.setAlarm(CIf.Info.intCtrlId,INT_TO_UINT(E_ALM_UMC.MotorError),0,ADR(SIf.Alm),E_AlmState.RST,CIf.Job.eMe_ActivAlmClass);
			me.StateMachine.intStateNext := Base_PLC.cSTA_ERROR;	
		END_IF
		
		IF (me.StateMachine.intStateNext <> Base_PLC.cSTA_ERROR) THEN
			// Reenter the RunBusy state again if the speed changes
			IF SIf.Par.uinSpeed_rpm <> SIf.Cur.uinSpeed_rpm THEN
				me.StateMachine.intStateNext := cSTA_RUNBusy;
			END_IF
			
			// Reenter the RunBusy state again if the direction changes.
			IF SIf.Par.eRotationDirection <> SIf.Cur.eDirection THEN
				me.StateMachine.intStateNext := cSTA_RUNBusy;
			END_IF

			CASE me.intCmd OF
				cCMD_Left:
					SIf.Par.eRotationDirection := E_TURN_DIRECTION.LEFT;
					me.StateMachine.intStateNext := cSTA_RUNBusy;
				cCMD_Right:
					SIf.Par.eRotationDirection := E_TURN_DIRECTION.RIGHT;
					me.StateMachine.intStateNext := cSTA_RUNBusy;
				BASE_PLC.cCMD_STOP:
					me.StateMachine.intStateNext := BASE_PLC.cSTA_STOPBusy;
			END_CASE
		END_IF
END_IF


//--------------------------------------------------------------------------------------
// Exit action
	IF (me.StateMachine.intState<>me.StateMachine.intStateNext) THEN
		;
	END_IF
END_METHOD

METHOD PROTECTED sta_RUNBusy : BOOL
VAR
	uniStatus 		: U_UMC_Lenze_Status;
END_VAR
// state implemetation
//--------------------------------------------------------------------------------------
// Entry action
	IF (me.StateMachine.intState<>me.StateMachine.intStateLastCycle) THEN
		me.StateMachine.intStateLastCycle := me.StateMachine.intState;

		SIf.Cur.uinSpeed_rpm := SIf.Par.uinSpeed_rpm;
		SIf.Cur.uinSpeedOuput := GetSpeedValue();
		SIf.Cur.eDirection 	:= SIf.Par.eRotationDirection;
		
		// Switch Motor ON
		IF SIf.Par.eRotationDirection < E_TURN_DIRECTION.MAX_E_TURN_DIRECTION THEN
			cmd_MotorOn(arTurnDirection[SIf.Par.eRotationDirection], SIf.Cur.uinSpeedOuput);
		ELSE
			pfbAlarmCtrl^.setAlarm(CIf.Info.intCtrlId,INT_TO_UINT(E_ALM_UMC.DirectionParameterOverflow),0,ADR(SIf.Alm),E_AlmState.RST,CIf.Job.eMe_ActivAlmClass);
			me.StateMachine.intStateNext := Base_PLC.cSTA_ERROR;	
		END_IF

		fbSimulationTimer.IN := FALSE;
		fbSimulationTimer.PT := UDINT_TO_TIME(SIf.Par.udiSimMotorOnTime_ms);
		fbSimulationTimer(); // set time/reset timer
		fbSimulationTimer.IN := TRUE; // start timer

	END_IF


//--------------------------------------------------------------------------------------
// Cyclic action
	IF (me.StateMachine.intState=me.StateMachine.intStateLastCycle) THEN
		IF (CIf.SwCfg.bolSimulation) THEN
			fbSimulationTimer(); // simulation time
			IF (fbSimulationTimer.Q) THEN
				SIf.In.uinMotorSetSpeed.intern 	:= SIf.Out.uinSpeedSetpoint.intern;
				SIf.In.uinMotorSetSpeed.intern 	:= SIf.Out.uinSpeedSetpoint.intern;
				uniStatus.Input 				:= 0;
				uniStatus.Data.DriveReady		:= 1;
				uniStatus.Data.SpeedActEqualSet := 1;
				uniStatus.Data.SpeedSetReached  := 1;
				uniStatus.Data.Status_1			:= 1;
				uniStatus.Data.Status_3			:= 1;
				uniStatus.Data.SpeedCcw			:= arTurnDirection[SIf.Par.eRotationDirection];
				SIf.In.uinStatus.intern 		:= uniStatus.Input;
			END_IF
		END_IF

		IF (me.StateMachine.udiTimeInState_ms > SIf.Par.udiMotorOnTime_ms) THEN
			pfbAlarmCtrl^.setAlarm(CIf.Info.intCtrlId,INT_TO_UINT(E_ALM_UMC.MotorOnTimeout),0,ADR(SIf.Alm),E_AlmState.RST,CIf.Job.eMe_ActivAlmClass);
			me.StateMachine.intStateNext := Base_PLC.cSTA_ERROR;	
		END_IF

		IF In_unStatus.Data.Trouble THEN
			pfbAlarmCtrl^.setAlarm(CIf.Info.intCtrlId,INT_TO_UINT(E_ALM_UMC.MotorError),0,ADR(SIf.Alm),E_AlmState.RST,CIf.Job.eMe_ActivAlmClass);
			me.StateMachine.intStateNext := Base_PLC.cSTA_ERROR;	
		END_IF
		
		IF (me.StateMachine.intStateNext <> Base_PLC.cSTA_ERROR) THEN
			IF (NOT In_unStatus.Data.Trouble) 
				AND (THIS^.arTurnDirection[SIf.Cur.eDirection] = In_unStatus.Data.SpeedCcw)	THEN
//				AND (In_unStatus.Data.SpeedSetReached) THEN
				me.StateMachine.intStateNext := cSTA_RUN;
			END_IF;	

			// Reenter the RunBusy state again if the speed changes
			IF GetSpeedValue() <> SIf.Cur.uinSpeedOuput THEN
				me.StateMachine.intStateLastCycle := -1;
			END_IF
			
			// Reenter the RunBusy state again if the direction changes.
			IF SIf.Par.eRotationDirection <> SIf.Cur.eDirection THEN
				me.StateMachine.intStateLastCycle := -1;
			END_IF
			
			CASE me.intCmd OF
				cCMD_Left:
					IF SIf.Par.eRotationDirection <> E_TURN_DIRECTION.LEFT THEN
						SIf.Par.eRotationDirection := E_TURN_DIRECTION.LEFT;
						me.StateMachine.intStateLastCycle := -1;
					END_IF
				cCMD_Right:
					IF SIf.Par.eRotationDirection <> E_TURN_DIRECTION.RIGHT THEN
						SIf.Par.eRotationDirection := E_TURN_DIRECTION.RIGHT;
						me.StateMachine.intStateLastCycle := -1;
					END_IF
				BASE_PLC.cCMD_STOP:
					me.StateMachine.intStateNext := BASE_PLC.cSTA_STOPBusy;
			END_CASE
		END_IF
END_IF


//--------------------------------------------------------------------------------------
// Exit action
	IF (me.StateMachine.intState<>me.StateMachine.intStateNext) THEN
		;
	END_IF
END_METHOD

METHOD PROTECTED sta_SETOPERATIONMODE : BOOL
VAR
	uinECatStatus		: UINT;

	fbEcReqSlaveState 	: FB_EcReqSlaveState;
	bExecute        	: BOOL;
	uinReqState     	: WORD := EC_DEVICE_STATE_OP;
	bError          	: BOOL;
	nErrId          	: UDINT;
END_VAR
// state implemetation
//--------------------------------------------------------------------------------------
// Entry action
	IF (me.StateMachine.intState<>me.StateMachine.intStateLastCycle) THEN
		me.StateMachine.intStateLastCycle := me.StateMachine.intState;
	END_IF


//--------------------------------------------------------------------------------------
// Cyclic action
	IF (me.StateMachine.intState=me.StateMachine.intStateLastCycle) THEN
		bExecute := NOT ((In_uinECATState AND cEtherCAT_MODE_MASK) = cEtherCAT_OP_MODE);

		IF NOT bExecute THEN
			me.StateMachine.intStateNext := UMC_CmdState.cSTA_RESETMOTORERROR;
		END_IF

		fbEcReqSlaveState(
			sNetId		:= F_CreateAmsNetId(In_strNetId), 
			nSlaveAddr	:= In_uintPort, 
			bExecute	:= bExecute, 
			state		:= uinReqState  );

		IF (me.StateMachine.udiTimeInState_ms > SIf.Par.udiStartupOnTime_ms) THEN
			pfbAlarmCtrl^.setAlarm(CIf.Info.intCtrlId,INT_TO_UINT(E_ALM_UMC.MotorError),0,ADR(SIf.Alm),E_AlmState.RST,CIf.Job.eMe_ActivAlmClass);
			me.StateMachine.intStateNext := Base_PLC.cSTA_ERROR;	
		END_IF
END_IF


//--------------------------------------------------------------------------------------
// Exit action
	IF (me.StateMachine.intState<>me.StateMachine.intStateNext) THEN
		Out_unControl.Data.ResetFault := FALSE;
	END_IF
END_METHOD

METHOD PROTECTED sta_STOP : BOOL
VAR_INPUT
END_VAR
// state implemetation
//--------------------------------------------------------------------------------------
// Entry action
	IF (me.StateMachine.intState<>me.StateMachine.intStateLastCycle) THEN
		me.StateMachine.intStateLastCycle := me.StateMachine.intState;

	END_IF


//--------------------------------------------------------------------------------------
// Cyclic action
	IF (me.StateMachine.intState=me.StateMachine.intStateLastCycle) THEN
		CASE me.intCmd OF
			cCMD_Left:
				SIf.Par.eRotationDirection := E_TURN_DIRECTION.LEFT;
				me.StateMachine.intStateNext := cSTA_RUNBusy;
			cCMD_Right:
				SIf.Par.eRotationDirection := E_TURN_DIRECTION.RIGHT;
				me.StateMachine.intStateNext := cSTA_RUNBusy;
			BASE_PLC.cCMD_RUN:
				me.StateMachine.intStateNext := cSTA_RUNBusy;
		END_CASE
	END_IF


//--------------------------------------------------------------------------------------
// Exit action
	IF (me.StateMachine.intState<>me.StateMachine.intStateNext) THEN
		;
	END_IF
END_METHOD

METHOD PROTECTED sta_STOPBusy : BOOL
VAR
	uniStatus 		: U_UMC_Lenze_Status;
END_VAR
// state implemetation
//--------------------------------------------------------------------------------------
// Entry action
	IF (me.StateMachine.intState<>me.StateMachine.intStateLastCycle) THEN
		me.StateMachine.intStateLastCycle := me.StateMachine.intState;
		// Switch Motor Off
		cmd_MotorStop();
	END_IF


//--------------------------------------------------------------------------------------
// Cyclic action
	IF (me.StateMachine.intState=me.StateMachine.intStateLastCycle) THEN
		IF (CIf.SwCfg.bolSimulation) THEN
			SIf.In.uinMotorSetSpeed.intern 	:= 0;
			SIf.In.intMotorActualSpeed.intern 	:= 0;
			uniStatus.Input 				:= 0;
			uniStatus.Data.ActSpeedIsZero	:= TRUE;
			SIf.In.uinStatus.intern 		:= uniStatus.Input;
		END_IF

		IF (me.StateMachine.udiTimeInState_ms < SIf.Par.udiMotorOnTime_ms) THEN
			IF (NOT In_unStatus.Data.Trouble) AND (In_unStatus.Data.ActSpeedIsZero) THEN
				me.StateMachine.intStateNext := Base_PLC.cSTA_STOP;
			END_IF;	
		ELSE
			pfbAlarmCtrl^.setAlarm(CIf.Info.intCtrlId,INT_TO_UINT(E_ALM_UMC.MotorError),0,ADR(SIf.Alm),E_AlmState.RST,CIf.Job.eMe_ActivAlmClass);
			me.StateMachine.intStateNext := Base_PLC.cSTA_ERROR;	
		END_IF
END_IF


//--------------------------------------------------------------------------------------
// Exit action
	IF (me.StateMachine.intState<>me.StateMachine.intStateNext) THEN
		Out_unControl.Data.ResetFault := FALSE;
	END_IF
END_METHOD

METHOD PROTECTED StateMachine : BOOL
SUPER^.StateMachine();

// main statemachine of base controller
CASE me.StateMachine.intState OF
	cSTA_RUNBusy:
		THIS^.sta_RUNBusy();
	cSTA_RUN:
		THIS^.sta_RUN();
	cSTA_STOPBusy: 
        THIS^.sta_STOPBusy();
    cSTA_STOP: 
        THIS^.sta_STOP();
	UMC_CmdState.cSTA_RESETMOTORERROR:
		THIS^.sta_RESETMOTORERROR();
	UMC_CmdState.cSTA_SETOPERATIONMODE:
		THIS^.sta_SETOPERATIONMODE();
END_CASE;
END_METHOD

END_FUNCTION_BLOCK

// POUs/Controller/Lvl0/VLV (Valve controller)/FB_VLV
FUNCTION_BLOCK FB_VLV EXTENDS FB_CtrlBase
VAR_INPUT
	In_bolOpened: BOOL;
	In_bolClosed: BOOL;
END_VAR
VAR_OUTPUT
	Out_bolOpen: BOOL;
	Out_bolClose: BOOL;
END_VAR
VAR
	/// Specific interface struct for public access
	SIf: T_Ctrl_SIf_VLV;
END_VAR

(*__________________________________________________________________________________________________
¦	
¦	Vistaprint Schweiz GmbH
¦	CH - 8401 Winterthur
¦
¦	www.vistaprint.ch - info@vistaprint.ch
¦___________________________________________________________________________________________________

Function desription:
Basic valve controller

History:
Version		Date			Author		Comment
---------------------------------------------------------------------------------------------------
0.00.1		06.03.2014		AVME/DSC	Start history. Based on CYL controller

___________________________________________________________________________________________________*)


SUPER^();

(*
IF (me.bolActivate) THEN // cyclic call enabled
	IF (CIf.Info.bolInitDone=FALSE) THEN // first cycle -> init
		CtrlInit();
		CIf.Info.bolInitDone := TRUE;
	ELSE
		CycleStartDuty();
	
		Always();
		
		StateMachine();
		
		CycleEndDuty();
	END_IF
END_IF;
*)

METHOD PROTECTED Always : BOOL
IF (me.bolChangeBackToAUTO=TRUE) THEN // switch mode to automatic switch off controller
	//me.StateMachine.intStateNext := cSTA_OFFBusy;
	me.bolChangeBackToAUTO := FALSE; // for valve no change to off when switch to automatic!!
END_IF

SUPER^.Always();

// ----------------------------------------------------------------------------------
// cyclic actions outside of statemachine
IF (me.StateMachine.intState<>cSTA_SINGLE_ANSWER) THEN
	
	; // always error supervision
	// ----------------------------------------------------------------------------------
	// overrule error always from base -> no EOFF State!! in EOFF go to OFF
	IF (me.StateMachine.intStateNext = cSTA_EOFFBusy) THEN
		IF (me.StateMachine.intState=cSTA_OFF) THEN
			me.StateMachine.intStateNext := cSTA_OFF;
		ELSE // stay in OFF
			me.StateMachine.intStateNext := cSTA_OFFBusy;
		END_IF
	END_IF
END_IF
END_METHOD

PROPERTY PUBLIC CtrlSIf : POINTER TO T_Ctrl_SIf_VLV
GET
CtrlSIf := ADR(SIf);
END_GET
END_PROPERTY

METHOD FB_init : BOOL
VAR_INPUT
	///if TRUE, the retain variables are initialized (warm start / cold start)
	bInitRetains: BOOL;
	///if TRUE, the instance afterwards gets moved into the copy code (online change)
	bInCopyCode: BOOL;
END_VAR
VAR
	ii: UINT;
END_VAR
//------------------------------------------------------------------------------------------------------------------------
// to manually change in new FUB implementation!!!
// define valid commands for this controller
FOR ii:= 0 TO (SIZEOF(CIf.Job.aCmdList)/SIZEOF(CIf.Job.aCmdList[0])-1) BY 1 DO
	IF (CIf.Job.aCmdList[ii].intCmd=cCMD_INITIALIZED) THEN
		// found first empty array element
		EXIT;
	END_IF
END_FOR

CIf.Job.aCmdList[ii].intCmd := cCMD_OPEN;
CIf.Job.aCmdList[ii].strName := 'Open';
CIf.Job.aCmdList[ii].bolAvailable := TRUE;
ii := ii +1;
CIf.Job.aCmdList[ii].intCmd := cCMD_CLOSE; 
CIf.Job.aCmdList[ii].strName := 'Close';
CIf.Job.aCmdList[ii].bolAvailable := TRUE;

// set name of class/typ
CIf.Info.strType := 'FB_VLV';
CIf.Info.strFullName := 'Valve Controller';

// set alarm class
SIf.Alm[E_ALM_VLV.SensorOpenAlwaysOn].eAlmClass := E_AlmClass.TSTOP;
SIf.Alm[E_ALM_VLV.SensorOpenAlwaysOn].strText := 'sensor open always on'; 
SIf.Alm[E_ALM_VLV.SensorOpenNotReached].eAlmClass := E_AlmClass.TSTOP;
SIf.Alm[E_ALM_VLV.SensorOpenNotReached].strText := 'timeout open - sensor open not reached';
SIf.Alm[E_ALM_VLV.SensorCloseAlwaysOn].eAlmClass := E_AlmClass.TSTOP;
SIf.Alm[E_ALM_VLV.SensorCloseAlwaysOn].strText := 'sensor close always on';
SIf.Alm[E_ALM_VLV.SensorCloseNotReached].eAlmClass := E_AlmClass.TSTOP;
SIf.Alm[E_ALM_VLV.SensorCloseNotReached].strText := 'timeout close - sensor close not reached';
SIf.Alm[E_ALM_VLV.InterlockOpen].eAlmClass := E_AlmClass.OFF;
SIf.Alm[E_ALM_VLV.InterlockOpen].strText := 'interlock open - movement stopped';
SIf.Alm[E_ALM_VLV.InterlockClose].eAlmClass := E_AlmClass.OFF;
SIf.Alm[E_ALM_VLV.InterlockClose].strText := 'interlock close - movement stopped';

//*******************************************************************************
// initial values
//*******************************************************************************

// Configuration defaults of class
CIf.SwCfg.bolExist := TRUE;
CIf.SwCfg.bolEnable := TRUE;
CIf.SwCfg.bolSimulation := FALSE;

// Parameter defaults of class
SIf.Par.udiOpenTime_ms := 4000;
SIf.Par.udiCloseTime_ms := 4000;
SIf.Par.udiSimOpenTime_ms := SIf.Par.udiOpenTime_ms/2;	
SIf.Par.udiSimCloseTime_ms := SIf.Par.udiCloseTime_ms/2;
END_METHOD

METHOD PROTECTED getCmdState : STRING
VAR_INPUT
	intCmdState: INT;
	bolState: BOOL;
END_VAR
getCmdState := SUPER^.getCmdState(intCmdState:=intCmdState,bolState:=bolState); // get global/base defined cmds/states
IF (getCmdState='') THEN // global not defined get local
	// get string cmd/state string information in runtime
	IF (bolState=FALSE) THEN
		// cmd's
		CASE intCmdState OF
			VLV_CmdState.cCMD_OPEN: 
				getCmdState := 'cCMD_OPEN';
			VLV_CmdState.cCMD_CLOSE: 
				getCmdState := 'cCMD_CLOSE';
		ELSE
			getCmdState := 'Cmd not defined';
		END_CASE;
	ELSE
	
	// cmd's
		CASE intCmdState OF
			VLV_CmdState.cSTA_OPENBusy: 
				getCmdState := 'cSTA_OPENBusy';
			VLV_CmdState.cSTA_OPEN: 
				getCmdState := 'cSTA_OPEN';
			VLV_CmdState.cSTA_CLOSEBusy: 
				getCmdState := 'cSTA_CLOSEBusy';
			VLV_CmdState.cSTA_CLOSE: 
				getCmdState := 'cSTA_CLOSE';
		ELSE
			getCmdState := 'State not defined';
		END_CASE;
	END_IF
END_IF
END_METHOD

METHOD getCtrlSIf : POINTER TO T_Ctrl_SIf_VLV
getCtrlSIf := ADR(SIf);
END_METHOD

METHOD PROTECTED IoInBridge : BOOL
// digitale and analoge inputs read from hardware or forcing
SIf.In.bolOpen.map := THIS^.In_bolOpened;
SIf.In.bolClose.map := THIS^.In_bolClosed;

IF (CIf.SwCfg.bolSimulation = FALSE) THEN
	getInBol(CIf.Job.bolIoForce,ADR(SIf.In.bolOpen));
	getInBol(CIf.Job.bolIoForce,ADR(SIf.In.bolClose));
ELSE
	//simulation of global IO
END_IF
END_METHOD

METHOD PROTECTED IoOutBridge : BOOL
VAR
	bolSwitchValvesOff: BOOL;
END_VAR
// digitale and analoge inputs read from hardware or forcing
IF (CIf.SwCfg.bolSimulation = FALSE) THEN
	setOutBol(CIf.Job.bolIoForce ,ADR(SIf.Out.bolOpen));
	setOutBol(CIf.Job.bolIoForce ,ADR(SIf.Out.bolClose));
	
	// check interlocks to prevent damages
	IF (CIf.Job.bolIlkOverwrite=FALSE) THEN
		bolSwitchValvesOff := FALSE;
		
		IF (SIf.Ilk.bolOpen=TRUE) THEN
			// switch off?
			IF (SIf.Cfg.eTyp = E_Typ_VLV.Valve1_Sensor0) OR (SIf.Cfg.eTyp = E_Typ_VLV.Valve1_Sensor2) 
				OR (SIf.Cfg.eTyp = E_Typ_VLV.Valve1_SensorOpened) OR (SIf.Cfg.eTyp = E_Typ_VLV.Valve1_SensorClosed) THEN
				// monostabil valve -> do nothing
			ELSE
				// bistable valve ->  switch both off
				bolSwitchValvesOff := TRUE;
				IF (SIf.Out.bolOpen.map=1) THEN
					pfbAlarmCtrl^.setAlarm(CIf.Info.intCtrlId,E_ALM_VLV.InterlockOpen,0,ADR(SIf.Alm),E_AlmState.RST,CIf.Job.eMe_ActivAlmClass);
				END_IF
			END_IF
		END_IF
		
		IF (SIf.Ilk.bolClose=TRUE) THEN
			// switch off?
			IF (SIf.Cfg.eTyp = E_Typ_VLV.Valve1_Sensor0) OR (SIf.Cfg.eTyp = E_Typ_VLV.Valve1_Sensor2) 
				OR (SIf.Cfg.eTyp = E_Typ_VLV.Valve1_SensorOpened) OR (SIf.Cfg.eTyp = E_Typ_VLV.Valve1_SensorClosed) THEN
				// monostabil valve -> do nothing
				;
			ELSE
				// bistable valve -> switch both off
				bolSwitchValvesOff := TRUE;
				IF (SIf.Out.bolClose.map=1) THEN
					pfbAlarmCtrl^.setAlarm(CIf.Info.intCtrlId,E_ALM_VLV.InterlockClose,0,ADR(SIf.Alm),E_AlmState.RST,CIf.Job.eMe_ActivAlmClass);
				END_IF;
			END_IF
		END_IF
		
		// bistable valve -> switch both off
		IF (bolSwitchValvesOff) THEN
			SIf.Out.bolOpen.map := FALSE;
			SIf.Out.bolClose.map := FALSE;
		END_IF
		
	END_IF

	THIS^.Out_bolOpen := SIf.Out.bolOpen.map;
	THIS^.Out_bolClose := SIf.Out.bolClose.map;
END_IF
END_METHOD

METHOD PROTECTED sta_CLOSE : BOOL
// state implemetation
//--------------------------------------------------------------------------------------
// Entry action
	IF (me.StateMachine.intState<>me.StateMachine.intStateLastCycle) THEN
		me.StateMachine.intStateLastCycle := me.StateMachine.intState;

	END_IF

//--------------------------------------------------------------------------------------
// Cyclic action
	IF (me.StateMachine.intState=me.StateMachine.intStateLastCycle) THEN

		// Simulation
		IF (CIf.SwCfg.bolSimulation) THEN
			;
		END_IF
		
		// State Change Condition
		IF (SIf.In.bolOpen.intern) THEN
			// sensor open always on
			pfbAlarmCtrl^.setAlarm(CIf.Info.intCtrlId,E_ALM_VLV.SensorOpenAlwaysOn,0,ADR(SIf.Alm),E_AlmState.RST,CIf.Job.eMe_ActivAlmClass);
			me.StateMachine.intStateNext :=  cSTA_ERROR;
		ELSIF ((SIf.In.bolClose.intern = FALSE) AND ((SIf.Cfg.eTyp = E_Typ_VLV.Valve1_SensorClosed) OR (SIf.Cfg.eTyp = E_Typ_VLV.Valve2_SensorClosed))) THEN // wait time until error?
			me.StateMachine.intStateNext := VLV_CmdState.cSTA_CLOSEBusy;
		ELSIF(me.intCmd=VLV_CmdState.cCMD_OPEN) THEN
			me.StateMachine.intStateNext := VLV_CmdState.cSTA_OPENBusy;
		END_IF
	END_IF

//--------------------------------------------------------------------------------------
// Exit action
	IF (me.StateMachine.intState<>me.StateMachine.intStateNext) THEN
		;
	END_IF
END_METHOD

METHOD PROTECTED sta_CLOSEBusy : BOOL
// state implemetation
//--------------------------------------------------------------------------------------
// Entry action
	IF (me.StateMachine.intState<>me.StateMachine.intStateLastCycle) THEN
		me.StateMachine.intStateLastCycle := me.StateMachine.intState;
		
		SIf.Out.bolOpen.intern := FALSE;
		SIf.Out.bolClose.intern := TRUE;
		
		fbSimulationTimer.IN := FALSE;
		fbSimulationTimer.PT := UDINT_TO_TIME(SIf.Par.udiSimCloseTime_ms);
		fbSimulationTimer(); // set time/reset timer
		fbSimulationTimer.IN := TRUE; // start timer
	END_IF


//--------------------------------------------------------------------------------------
// Cyclic action
	IF (me.StateMachine.intState=me.StateMachine.intStateLastCycle) THEN

		// Simulation
		IF (CIf.SwCfg.bolSimulation) THEN
			fbSimulationTimer(); // simulation time
			IF (fbSimulationTimer.Q) THEN
				SIf.In.bolClose.intern := TRUE;
				SIf.In.bolOpen.intern := FALSE;
			END_IF
		END_IF
		
		// State Change Condition
		IF (me.StateMachine.udiTimeInState_ms>SIf.Par.udiCloseTime_ms) THEN
			IF (SIf.In.bolOpen.intern) THEN
				// sensor open always on 
				pfbAlarmCtrl^.setAlarm(CIf.Info.intCtrlId,E_ALM_VLV.SensorOpenAlwaysOn,0,ADR(SIf.Alm),E_AlmState.RST,CIf.Job.eMe_ActivAlmClass);
			ELSE
				// timeout close valve
				pfbAlarmCtrl^.setAlarm(CIf.Info.intCtrlId,E_ALM_VLV.SensorCloseNotReached,0,ADR(SIf.Alm),E_AlmState.RST,CIf.Job.eMe_ActivAlmClass);
			END_IF
			me.StateMachine.intStateNext :=  cSTA_ERROR;
		ELSIF (SIf.In.bolClose.intern) AND(SIf.In.bolOpen.intern=FALSE) THEN
			me.StateMachine.intStateNext := VLV_CmdState.cSTA_CLOSE;
		ELSIF ((SIf.Cfg.eTyp = E_Typ_VLV.Valve1_SensorOpened) OR (SIf.Cfg.eTyp = E_Typ_VLV.Valve2_SensorOpened))
				 AND (SIf.In.bolOpen.intern=FALSE) AND (me.StateMachine.udiTimeInState_ms>SIf.Par.udiSimCloseTime_ms) THEN
			me.StateMachine.intStateNext := VLV_CmdState.cSTA_CLOSE;
		ELSIF ((SIf.Cfg.eTyp = E_Typ_VLV.Valve1_Sensor0) OR (SIf.Cfg.eTyp = E_Typ_VLV.Valve2_Sensor0))
				AND (me.StateMachine.udiTimeInState_ms>SIf.Par.udiSimCloseTime_ms) THEN
			me.StateMachine.intStateNext := VLV_CmdState.cSTA_CLOSE;		
		ELSIF(me.intCmd=VLV_CmdState.cCMD_OPEN) THEN
			me.StateMachine.intStateNext := VLV_CmdState.cSTA_OPENBusy;
		END_IF
	END_IF


//--------------------------------------------------------------------------------------
// Exit action
	IF (me.StateMachine.intState<>me.StateMachine.intStateNext) THEN
		SIf.Cur.udiMoveTimeClose := me.StateMachine.udiTimeInState_ms;
	END_IF
END_METHOD

METHOD PROTECTED sta_ERROR : BOOL
// state implemetation
//--------------------------------------------------------------------------------------
// Entry action
	IF (me.StateMachine.intState<>me.StateMachine.intStateLastCycle) THEN
		me.StateMachine.intStateHistory := me.StateMachine.intStateLastCycle; // -> possibillity to go back to state before error
		me.StateMachine.intStateLastCycle := me.StateMachine.intState;
		
	END_IF

//--------------------------------------------------------------------------------------
// Cyclic action
	IF (me.StateMachine.intState=me.StateMachine.intStateLastCycle) THEN
		
		;	
		// State Change Condition
		IF (CIf.Job.bolAlmReset = TRUE) THEN
			me.StateMachine.intStateNext := cSTA_ERRORQuit;
		END_IF
	END_IF

//--------------------------------------------------------------------------------------
// Exit action
	IF (me.StateMachine.intState<>me.StateMachine.intStateNext) THEN
		;
	END_IF
END_METHOD

METHOD PROTECTED sta_ERRORQuit : BOOL
// state implemetation
//--------------------------------------------------------------------------------------
// Entry action
	IF (me.StateMachine.intState<>me.StateMachine.intStateLastCycle) THEN
		me.StateMachine.intStateLastCycle := me.StateMachine.intState;
		
	END_IF


//--------------------------------------------------------------------------------------
// Cyclic action
	IF (me.StateMachine.intState=me.StateMachine.intStateLastCycle) THEN
		
		;
		// evtl. wait time if reset of device is necessary and then decide to go to states or ERROR state
		IF (CIf.Job.bolAlmReset = TRUE) THEN
			CIf.Job.eMe_ActivAlmClass := E_AlmClass.NONE; // reset feedback channel for parent
			CIf.Job.bolAlmReset := FALSE;
		END_IF
		
		// State Change Condition
		IF (CIf.Job.bolAlmReset = FALSE) THEN
			IF (me.StateMachine.intStateHistory<=cSTA_PON) THEN
				me.StateMachine.intStateNext := cSTA_PONBusy;
			ELSIF(me.intCmd=cCMD_OFF) THEN
				me.StateMachine.intStateNext := cSTA_OFFBusy;
			ELSIF(me.intCmd=VLV_CmdState.cCMD_OPEN) THEN
				me.StateMachine.intStateNext := VLV_CmdState.cSTA_OPENBusy;
			ELSIF(me.intCmd=VLV_CmdState.cCMD_CLOSE) THEN
				me.StateMachine.intStateNext := VLV_CmdState.cSTA_CLOSEBusy;
			END_IF
		END_IF
	END_IF


//--------------------------------------------------------------------------------------
// Exit action
	IF (me.StateMachine.intState<>me.StateMachine.intStateNext) THEN
		;
	END_IF
END_METHOD

METHOD PROTECTED sta_OFF : BOOL
// state implemetation
//--------------------------------------------------------------------------------------
// Entry action
	IF (me.StateMachine.intState<>me.StateMachine.intStateLastCycle) THEN
		me.StateMachine.intStateLastCycle := me.StateMachine.intState;
		
	END_IF


//--------------------------------------------------------------------------------------
// Cyclic action
	IF (me.StateMachine.intState=me.StateMachine.intStateLastCycle) THEN
		
		;
		
		// State Change Condition
		IF (me.Alarm.eActivAlmClass<>E_AlmClass.EOFF) AND (me.Alarm.eActivAlmClass<>E_AlmClass.OFF) THEN
			IF (me.intCmd=VLV_CmdState.cCMD_OPEN) THEN 
				me.StateMachine.intStateNext := VLV_CmdState.cSTA_OPENBusy;
			ELSIF(me.intCmd=VLV_CmdState.cCMD_CLOSE) THEN
				me.StateMachine.intStateNext := VLV_CmdState.cSTA_CLOSEBusy;
			END_IF
		END_IF
	END_IF




//--------------------------------------------------------------------------------------
// Exit action
	IF (me.StateMachine.intState<>me.StateMachine.intStateNext) THEN
		;
	END_IF
END_METHOD

METHOD PROTECTED sta_OFFBusy : BOOL
// state implemetation
//--------------------------------------------------------------------------------------
// Entry action
	IF (me.StateMachine.intState<>me.StateMachine.intStateLastCycle) THEN
		me.StateMachine.intStateLastCycle := me.StateMachine.intState;
		
	END_IF


//--------------------------------------------------------------------------------------
// Cyclic action
	IF (me.StateMachine.intState=me.StateMachine.intStateLastCycle) THEN
		
		// switch off?
		IF (SIf.Cfg.eTyp = E_Typ_VLV.Valve1_Sensor0) OR (SIf.Cfg.eTyp = E_Typ_VLV.Valve1_Sensor2) 
			OR (SIf.Cfg.eTyp = E_Typ_VLV.Valve1_SensorOpened) OR (SIf.Cfg.eTyp = E_Typ_VLV.Valve1_SensorClosed) THEN
			// monostabil valve -> do nothing
			;
		ELSE
			// bistable valve -> switch both off
			SIf.Out.bolOpen.intern := FALSE;
			SIf.Out.bolClose.intern := FALSE;
		END_IF
		
		
		
		// State Change Condition
		IF (TRUE) THEN
			me.StateMachine.intStateNext := cSTA_OFF;
		END_IF
	END_IF




//--------------------------------------------------------------------------------------
// Exit action
	IF (me.StateMachine.intState<>me.StateMachine.intStateNext) THEN
		;
	END_IF
END_METHOD

METHOD PROTECTED sta_OPEN : BOOL
// state implemetation
//--------------------------------------------------------------------------------------
// Entry action
	IF (me.StateMachine.intState<>me.StateMachine.intStateLastCycle) THEN
		me.StateMachine.intStateLastCycle := me.StateMachine.intState;

	END_IF

//--------------------------------------------------------------------------------------
// Cyclic action
	IF (me.StateMachine.intState=me.StateMachine.intStateLastCycle) THEN

		// Simulation
		IF (CIf.SwCfg.bolSimulation) THEN
			;
		END_IF
		
		// State Change Condition
		IF (SIf.In.bolClose.intern) THEN
			// sensor close always on
			pfbAlarmCtrl^.setAlarm(CIf.Info.intCtrlId,E_ALM_VLV.SensorCloseAlwaysOn,0,ADR(SIf.Alm),E_AlmState.RST,CIf.Job.eMe_ActivAlmClass);
			me.StateMachine.intStateNext :=  cSTA_ERROR;
		ELSIF ((SIf.In.bolOpen.intern = FALSE) AND ((SIf.Cfg.eTyp = E_Typ_VLV.Valve1_SensorOpened) OR (SIf.Cfg.eTyp = E_Typ_VLV.Valve2_SensorOpened))) THEN // wait time until error?
			me.StateMachine.intStateNext := VLV_CmdState.cSTA_OPENBusy;
		ELSIF(me.intCmd=VLV_CmdState.cCMD_CLOSE) THEN
			me.StateMachine.intStateNext := VLV_CmdState.cSTA_CLOSEBusy;
		END_IF
	END_IF

//--------------------------------------------------------------------------------------
// Exit action
	IF (me.StateMachine.intState<>me.StateMachine.intStateNext) THEN
		;
	END_IF
END_METHOD

METHOD PROTECTED sta_OPENBusy : BOOL
// state implemetation
//--------------------------------------------------------------------------------------
// Entry action
	IF (me.StateMachine.intState<>me.StateMachine.intStateLastCycle) THEN
		me.StateMachine.intStateLastCycle := me.StateMachine.intState;

		SIf.Out.bolOpen.intern := TRUE;
		SIf.Out.bolClose.intern := FALSE;
		
		fbSimulationTimer.IN := FALSE;
		fbSimulationTimer.PT := UDINT_TO_TIME(SIf.Par.udiSimOpenTime_ms);
		fbSimulationTimer(); // set time/reset timer
		fbSimulationTimer.IN := TRUE; // start timer
	END_IF


//--------------------------------------------------------------------------------------
// Cyclic action
	IF (me.StateMachine.intState=me.StateMachine.intStateLastCycle) THEN

		// Simulation
		IF (CIf.SwCfg.bolSimulation) THEN
			fbSimulationTimer(); // simulation time
			IF (fbSimulationTimer.Q) THEN
				SIf.In.bolOpen.intern := TRUE;
				SIf.In.bolClose.intern := FALSE;
			END_IF
		END_IF
		
		// State Change Condition
		IF (me.StateMachine.udiTimeInState_ms > SIf.Par.udiOpenTime_ms) THEN
			IF (SIf.In.bolClose.intern) THEN
				// sensor close always on
				pfbAlarmCtrl^.setAlarm(CIf.Info.intCtrlId,E_ALM_VLV.SensorCloseAlwaysOn,0,ADR(SIf.Alm),E_AlmState.RST,CIf.Job.eMe_ActivAlmClass);
			ELSE
				// timeout open valve
				pfbAlarmCtrl^.setAlarm(CIf.Info.intCtrlId,E_ALM_VLV.SensorOpenNotReached,0,ADR(SIf.Alm),E_AlmState.RST,CIf.Job.eMe_ActivAlmClass);
			END_IF
			me.StateMachine.intStateNext :=  cSTA_ERROR;
		ELSIF (SIf.In.bolOpen.intern) AND (SIf.In.bolClose.intern=FALSE) THEN
			me.StateMachine.intStateNext := VLV_CmdState.cSTA_OPEN;
		ELSIF ((SIf.Cfg.eTyp = E_Typ_VLV.Valve1_SensorClosed) OR (SIf.Cfg.eTyp = E_Typ_VLV.Valve2_SensorClosed))
				 AND (SIf.In.bolClose.intern=FALSE) AND (me.StateMachine.udiTimeInState_ms>SIf.Par.udiSimOpenTime_ms) THEN
			me.StateMachine.intStateNext := VLV_CmdState.cSTA_OPEN;
		ELSIF ((SIf.Cfg.eTyp = E_Typ_VLV.Valve1_Sensor0) OR (SIf.Cfg.eTyp = E_Typ_VLV.Valve2_Sensor0))
				AND (me.StateMachine.udiTimeInState_ms>SIf.Par.udiSimOpenTime_ms) THEN
			me.StateMachine.intStateNext := VLV_CmdState.cSTA_OPEN;		
		ELSIF(me.intCmd=VLV_CmdState.cCMD_CLOSE) THEN
			me.StateMachine.intStateNext := VLV_CmdState.cSTA_CLOSEBusy;
		END_IF
	END_IF

//--------------------------------------------------------------------------------------
// Exit action
	IF (me.StateMachine.intState<>me.StateMachine.intStateNext) THEN
		SIf.Cur.udiMoveTimeOpen := me.StateMachine.udiTimeInState_ms;
	END_IF
END_METHOD

METHOD PROTECTED StateMachine : BOOL
SUPER^.StateMachine();

// main statemachine of base controller
CASE me.StateMachine.intState OF
    VLV_CmdState.cSTA_OPENBusy: 
        THIS^.sta_OPENBusy();
    VLV_CmdState.cSTA_OPEN: 
        THIS^.sta_OPEN();
    VLV_CmdState.cSTA_CLOSEBusy: 
        THIS^.sta_CLOSEBusy();
    VLV_CmdState.cSTA_CLOSE: 
        THIS^.sta_CLOSE();
END_CASE;
END_METHOD

END_FUNCTION_BLOCK

// POUs/Controller/Lvl0/VPC [Vacuum Pump Controller]/FB_VPC
FUNCTION_BLOCK FB_VPC EXTENDS FB_CtrlBase
VAR_INPUT
	In_bolVacuumOk			: BOOL;
	In_bolPumpOk			: BOOL;
END_VAR
VAR_OUTPUT
	Out_bolVaccumPumpOn		: BOOL;
END_VAR
VAR
	/// Specific interface struct for public access
	SIf					: T_Ctrl_SIf_VPC;
END_VAR

(*__________________________________________________________________________________________________
¦	
¦	Vistaprint Schweiz GmbH
¦	CH - 8401 Winterthur
¦
¦	www.vistaprint.ch - info@vistaprint.ch
¦___________________________________________________________________________________________________

Function desription:
Vacuum Pump implementation. 


History:
Version		Date			Author		Comment
---------------------------------------------------------------------------------------------------
0.00.1		09.07.2013		PC			Start history
___________________________________________________________________________________________________*)


SUPER^();

(*
IF (me.bolActivate) THEN // cyclic call enabled
	IF (CIf.Info.bolInitDone=FALSE) THEN // first cycle -> init
		CtrlInit();
		CIf.Info.bolInitDone := TRUE;
	ELSE
		CycleStartDuty();
	
		Always();
		
		StateMachine();
		
		CycleEndDuty();
	END_IF
END_IF;
*)

METHOD PROTECTED Always : BOOL
SUPER^.Always();

// ----------------------------------------------------------------------------------
// cyclic actions outside of statemachine
IF (me.StateMachine.intState<>cSTA_SINGLE_ANSWER) THEN
	
	; // always error supervision
	
END_IF

// ----------------------------------------------------------------------------------
// Conditions Always
IF (((me.Alarm.eActivAlmClass=E_AlmClass.EOFF) OR (me.Alarm.eActivAlmClass=E_AlmClass.OFF) OR (me.intCmd=cCMD_OFF))
		 AND (me.StateMachine.intState<>cSTA_ERROR) AND (me.StateMachine.intState<>cSTA_ERRORQuit) AND
		(me.StateMachine.intState<>cSTA_OFF) AND (me.StateMachine.intState<>cSTA_OFFBusy)) THEN
	// alarm evt EOFF, OFF or cmd off
	me.StateMachine.intStateNext := cSTA_OFFBusy;
END_IF
END_METHOD

PROPERTY PUBLIC CtrlSIf : POINTER TO T_Ctrl_SIf_VPC
GET
CtrlSIf := ADR(SIf);
END_GET
END_PROPERTY

METHOD FB_init : BOOL
VAR_INPUT
	bInitRetains : BOOL; // if TRUE, the retain variables are initialized (warm start / cold start)
	bInCopyCode : BOOL;  // if TRUE, the instance afterwards gets moved into the copy code (online change)
END_VAR
VAR
	iIdx		: UINT;
	iLength		: UINT;	
END_VAR
//------------------------------------------------------------------------------------------------------------------------
// to manually change in new FUB implementation!!!
// define valid commands for this controller
iLength := SIZEOF(CIf.Job.aCmdList)/SIZEOF(CIf.Job.aCmdList[0]);
iIdx := 0;

WHILE (iIdx < iLength) AND (CIf.Job.aCmdList[iIdx].intCmd <> cCMD_INITIALIZED) DO
	iIdx := iIdx + 1; 
END_WHILE

IF (iIdx < iLength) THEN
// Add configuration of own comands	
	CIf.Job.aCmdList[iIdx].intCmd := BASE_PLC.cCMD_RUN;
	CIf.Job.aCmdList[iIdx].strName := 'RUN'; 
	CIf.Job.aCmdList[iIdx].bolAvailable := TRUE;
ELSE
	// Error if the aCmdList Array is to small
END_IF

// set name of class/typ
CIf.Info.strType := 'FB_VPC';
CIf.Info.strFullName := 'Vacuum Pump Controller';

// set alarm class
SIf.Alm[E_ALM_VPC.VacuumPumpOnTimeout].eAlmClass := E_AlmClass.TSTOP;
SIf.Alm[E_ALM_VPC.VacuumPumpOnTimeout].strText := 'Vacuum pump On timeout'; 
SIf.Alm[E_ALM_VPC.VacuumPumpOffTimeout].eAlmClass := E_AlmClass.TSTOP;
SIf.Alm[E_ALM_VPC.VacuumPumpOffTimeout].strText := 'Vacuum pump Off timeout';
SIf.Alm[E_ALM_VPC.VacuumFailure].eAlmClass := E_AlmClass.TSTOP;
SIf.Alm[E_ALM_VPC.VacuumFailure].strText := 'Vacuum failure';

//*******************************************************************************
// initial values
//*******************************************************************************

// software configuration
CIf.SwCfg.bolExist := TRUE;
CIf.SwCfg.bolEnable := TRUE;
CIf.SwCfg.bolSimulation := FALSE;

// parameter
SIf.Par.udiVacuumPumpTime_ms := 10000;
SIf.Par.udiVacuumStabilizationTime_ms := 3000;
SIf.Par.udiSimVacuumPumpOnTime_ms := SIf.Par.udiVacuumPumpTime_ms / 2;
END_METHOD

METHOD PROTECTED getCmdState : STRING

VAR_INPUT
	intCmdState: INT;
	bolState: BOOL;
END_VAR
getCmdState := SUPER^.getCmdState(intCmdState:=intCmdState,bolState:=bolState); // get global/base defined cmds/states

IF (getCmdState='') THEN // global not defined get local
	// get string cmd/state string information in runtime
	IF (bolState=FALSE) THEN
		;// Comands's
	ELSE
		// States's
		CASE intCmdState OF
			VPC_CmdState.cSTA_VPC_StabilizeBusy: 
				getCmdState := 'cSTA_StabilizeBusy';
		END_CASE;
	END_IF
END_IF
END_METHOD

METHOD getCtrlSIf : POINTER TO T_Ctrl_SIf_VPC
getCtrlSIf := ADR(SIf);
END_METHOD

METHOD PROTECTED IoInBridge : BOOL
// digitale and analoge inputs read from hardware or forcing
SIf.In.bolVacuumOk.map := THIS^.In_bolVacuumOk;
SIf.In.bolPumpOn.map := THIS^.In_bolPumpOk;

IF (CIf.SwCfg.bolSimulation = FALSE) THEN
	getInBol(CIf.Job.bolIoForce,ADR(SIf.In.bolVacuumOk));
	getInBol(CIf.Job.bolIoForce,ADR(SIf.In.bolPumpOn));
ELSE
	//simulation of global IO
END_IF
END_METHOD

METHOD PROTECTED IoOutBridge : BOOL
VAR
	bolSwitchValvesOff: BOOL;
END_VAR
// digitale and analoge inputs read from hardware or forcing
IF (CIf.SwCfg.bolSimulation = FALSE) THEN
	setOutBol(CIf.Job.bolIoForce ,ADR(SIf.Out.bolVacuumPumpOn));

	THIS^.Out_bolVaccumPumpOn := SIf.Out.bolVacuumPumpOn.map;
END_IF
END_METHOD

METHOD PROTECTED sta_ERROR : BOOL
// state implemetation
//--------------------------------------------------------------------------------------
// Entry action
	IF (me.StateMachine.intState<>me.StateMachine.intStateLastCycle) THEN
		me.StateMachine.intStateHistory := me.StateMachine.intStateLastCycle; // -> possibillity to go back to state before error
		me.StateMachine.intStateLastCycle := me.StateMachine.intState;
		
	END_IF


//--------------------------------------------------------------------------------------
// Cyclic action
	IF (me.StateMachine.intState=me.StateMachine.intStateLastCycle) THEN
		
		;
		
		
		// State Change Condition
		IF (CIf.Job.bolAlmReset = TRUE) THEN
			me.StateMachine.intStateNext := cSTA_ERRORQuit;
		END_IF
	END_IF




//--------------------------------------------------------------------------------------
// Exit action
	IF (me.StateMachine.intState<>me.StateMachine.intStateNext) THEN
		;
	END_IF
END_METHOD

METHOD PROTECTED sta_ERRORQuit : BOOL
// state implemetation
//--------------------------------------------------------------------------------------
// Entry action
	IF (me.StateMachine.intState<>me.StateMachine.intStateLastCycle) THEN
		me.StateMachine.intStateLastCycle := me.StateMachine.intState;
		
	END_IF


//--------------------------------------------------------------------------------------
// Cyclic action
	IF (me.StateMachine.intState=me.StateMachine.intStateLastCycle) THEN
		
		;
		// evtl. wait time if reset of device is necessary and then decide to go to states or ERROR state
		IF (CIf.Job.bolAlmReset = TRUE) THEN
			CIf.Job.eMe_ActivAlmClass := E_AlmClass.NONE; // reset feedback channel for parent
			CIf.Job.bolAlmReset := FALSE;
		END_IF
		
		// State Change Condition
		IF (CIf.Job.bolAlmReset = FALSE) THEN
			IF (me.StateMachine.intStateHistory<=cSTA_PON) THEN
				me.StateMachine.intStateNext := cSTA_PONBusy;
			ELSIF(me.intCmd=cCMD_OFF) THEN
				me.StateMachine.intStateNext := cSTA_OFFBusy;
			ELSIF(me.intCmd=cCMD_STOP) THEN
				me.StateMachine.intStateNext := cSTA_STOPBusy;
			ELSIF(me.intCmd=BASE_PLC.cCMD_RUN) THEN
				me.StateMachine.intStateNext := BASE_PLC.cSTA_RUNBusy;
			END_IF
		END_IF
	END_IF




//--------------------------------------------------------------------------------------
// Exit action
	IF (me.StateMachine.intState<>me.StateMachine.intStateNext) THEN
		;
	END_IF
END_METHOD

METHOD PROTECTED sta_OFF : BOOL
VAR_INPUT
END_VAR
// state implemetation
//--------------------------------------------------------------------------------------
// Entry action
	IF (me.StateMachine.intState<>me.StateMachine.intStateLastCycle) THEN
		me.StateMachine.intStateLastCycle := me.StateMachine.intState;

	END_IF


//--------------------------------------------------------------------------------------
// Cyclic action
	IF (me.StateMachine.intState=me.StateMachine.intStateLastCycle) THEN
		IF me.intCmd = BASE_PLC.cCMD_RUN THEN
			me.StateMachine.intStateNext := BASE_PLC.cSTA_RUNBusy;
		END_IF
	END_IF


//--------------------------------------------------------------------------------------
// Exit action
	IF (me.StateMachine.intState<>me.StateMachine.intStateNext) THEN
		;
	END_IF
END_METHOD

METHOD PROTECTED sta_OFFBusy : BOOL
VAR_INPUT
END_VAR
// state implemetation
//--------------------------------------------------------------------------------------
// Entry action
	IF (me.StateMachine.intState<>me.StateMachine.intStateLastCycle) THEN
		me.StateMachine.intStateLastCycle := me.StateMachine.intState;
		// Switch Pump Off
		SIf.Out.bolVacuumPumpOn.intern := FALSE;
	END_IF


//--------------------------------------------------------------------------------------
// Cyclic action
	IF (me.StateMachine.intState=me.StateMachine.intStateLastCycle) THEN
		IF (CIf.SwCfg.bolSimulation) THEN
			SIf.In.bolPumpOn.intern := FALSE;
			SIf.In.bolVacuumOk.intern := FALSE;
		END_IF

		IF ((NOT SIf.In.bolPumpOn.intern) OR (NOT SIf.Cfg.VacuumPumpFeedback)) AND ((NOT SIf.In.bolVacuumOk.intern) OR (NOT SIf.Cfg.VacuumSensorAvailable)) THEN
			me.StateMachine.intStateNext := BASE_PLC.cSTA_OFF;
		END_IF;	
	END_IF


//--------------------------------------------------------------------------------------
// Exit action
	IF (me.StateMachine.intState<>me.StateMachine.intStateNext) THEN
		;
	END_IF
END_METHOD

METHOD PROTECTED sta_PON : BOOL
VAR_INPUT
END_VAR
// state implemetation
//--------------------------------------------------------------------------------------
// Entry action
	IF (me.StateMachine.intState<>me.StateMachine.intStateLastCycle) THEN
		me.StateMachine.intStateLastCycle := me.StateMachine.intState;
		
	END_IF


//--------------------------------------------------------------------------------------
// Cyclic action
	IF (me.StateMachine.intState=me.StateMachine.intStateLastCycle) THEN
		;
	END_IF




//--------------------------------------------------------------------------------------
// Exit action
	IF (me.StateMachine.intState<>me.StateMachine.intStateNext) THEN
		;
	END_IF
END_METHOD

METHOD PROTECTED sta_RUN : BOOL
VAR_INPUT
END_VAR
// state implemetation
//--------------------------------------------------------------------------------------
// Entry action
	IF (me.StateMachine.intState<>me.StateMachine.intStateLastCycle) THEN
		me.StateMachine.intStateLastCycle := me.StateMachine.intState;
	END_IF


//--------------------------------------------------------------------------------------
// Cyclic action
	IF (me.StateMachine.intState=me.StateMachine.intStateLastCycle) THEN
		// State Change Condition
		IF (NOT SIf.In.bolPumpOn.intern) AND (SIf.Cfg.VacuumPumpFeedback) THEN
			pfbAlarmCtrl^.setAlarm(CIf.Info.intCtrlId,INT_TO_UINT(E_ALM_VPC.VacuumPumpOnTimeout),0,ADR(SIf.Alm),E_AlmState.RST,CIf.Job.eMe_ActivAlmClass);
			me.StateMachine.intStateNext :=  BASE_PLC.cSTA_ERROR;
		END_IF;

		IF ((NOT SIf.In.bolVacuumOk.intern) AND (SIf.Cfg.VacuumSensorAvailable)) THEN
			pfbAlarmCtrl^.setAlarm(CIf.Info.intCtrlId,INT_TO_UINT(E_ALM_VPC.VacuumFailure),0,ADR(SIf.Alm),E_AlmState.RST,CIf.Job.eMe_ActivAlmClass);
			me.StateMachine.intStateNext :=  BASE_PLC.cSTA_ERROR;
		END_IF;	
	END_IF


//--------------------------------------------------------------------------------------
// Exit action
	IF (me.StateMachine.intState<>me.StateMachine.intStateNext) THEN
		;
	END_IF
END_METHOD

METHOD PROTECTED sta_RUNBusy : BOOL
VAR_INPUT
END_VAR
// state implemetation
//--------------------------------------------------------------------------------------
// Entry action
	IF (me.StateMachine.intState<>me.StateMachine.intStateLastCycle) THEN
		me.StateMachine.intStateLastCycle := me.StateMachine.intState;
		SIf.Out.bolVacuumPumpOn.intern := TRUE;

		fbSimulationTimer.IN := FALSE;
		fbSimulationTimer.PT := UDINT_TO_TIME(SIf.Par.udiSimVacuumPumpOnTime_ms);
		fbSimulationTimer(); // set time/reset timer
		fbSimulationTimer.IN := TRUE; // start timer
	END_IF


//--------------------------------------------------------------------------------------
// Cyclic action
	IF (me.StateMachine.intState=me.StateMachine.intStateLastCycle) THEN
		// Simulation
		IF (CIf.SwCfg.bolSimulation) THEN
			fbSimulationTimer(); // simulation time
			IF (fbSimulationTimer.Q) THEN
				SIf.In.bolPumpOn.intern := TRUE;
				SIf.In.bolVacuumOk.intern := TRUE;
			END_IF
		END_IF

		IF ((SIf.In.bolVacuumOk.intern) OR (NOT SIf.Cfg.VacuumPumpFeedback)) AND ((SIf.In.bolVacuumOk.intern) OR (NOT SIf.Cfg.VacuumSensorAvailable)) THEN
			me.StateMachine.intStateNext := VPC_CmdState.cSTA_VPC_StabilizeBusy;
		END_IF;		
		
		IF (me.StateMachine.udiTimeInState_ms > SIf.Par.udiVacuumPumpTime_ms) THEN
			IF (NOT SIf.In.bolPumpOn.intern) AND (SIf.Cfg.VacuumPumpFeedback) THEN
				pfbAlarmCtrl^.setAlarm(CIf.Info.intCtrlId,INT_TO_UINT(E_ALM_VPC.VacuumPumpOnTimeout),0,ADR(SIf.Alm),E_AlmState.RST,CIf.Job.eMe_ActivAlmClass);
			END_IF;

			IF ((NOT SIf.In.bolVacuumOk.intern) AND (SIf.Cfg.VacuumSensorAvailable)) THEN
				pfbAlarmCtrl^.setAlarm(CIf.Info.intCtrlId,INT_TO_UINT(E_ALM_VPC.VacuumFailure),0,ADR(SIf.Alm),E_AlmState.RST,CIf.Job.eMe_ActivAlmClass);
			END_IF;	

			me.StateMachine.intStateNext :=  cSTA_ERROR;
		END_IF
	END_IF


//--------------------------------------------------------------------------------------
// Exit action
	IF (me.StateMachine.intState<>me.StateMachine.intStateNext) THEN
		;
	END_IF
END_METHOD

METHOD PROTECTED sta_StabilizeVacuum : BOOL
VAR_INPUT
END_VAR
// state implemetation
//--------------------------------------------------------------------------------------
// Entry action
	IF (me.StateMachine.intState<>me.StateMachine.intStateLastCycle) THEN
		me.StateMachine.intStateLastCycle := me.StateMachine.intState;
	END_IF


//--------------------------------------------------------------------------------------
// Cyclic action
	IF (me.StateMachine.intState=me.StateMachine.intStateLastCycle) THEN
		// State Change Condition
		
		IF (me.StateMachine.udiTimeInState_ms > SIf.Par.udiVacuumStabilizationTime_ms) THEN
			me.StateMachine.intStateNext :=  BASE_PLC.cSTA_RUN;
		END_IF;	

		IF (NOT SIf.In.bolPumpOn.intern) AND (SIf.Cfg.VacuumPumpFeedback) THEN
			pfbAlarmCtrl^.setAlarm(CIf.Info.intCtrlId,INT_TO_UINT(E_ALM_VPC.VacuumPumpOnTimeout),0,ADR(SIf.Alm),E_AlmState.RST,CIf.Job.eMe_ActivAlmClass);
			me.StateMachine.intStateNext :=  BASE_PLC.cSTA_ERROR;
		END_IF;

		IF ((NOT SIf.In.bolVacuumOk.intern) AND (SIf.Cfg.VacuumSensorAvailable)) THEN
			pfbAlarmCtrl^.setAlarm(CIf.Info.intCtrlId,INT_TO_UINT(E_ALM_VPC.VacuumFailure),0,ADR(SIf.Alm),E_AlmState.RST,CIf.Job.eMe_ActivAlmClass);
			me.StateMachine.intStateNext :=  BASE_PLC.cSTA_ERROR;
		END_IF;	
	END_IF


//--------------------------------------------------------------------------------------
// Exit action
	IF (me.StateMachine.intState<>me.StateMachine.intStateNext) THEN
		;
	END_IF
END_METHOD

METHOD PROTECTED StateMachine : BOOL
SUPER^.StateMachine();

// main statemachine of base controller
CASE me.StateMachine.intState OF
    VPC_CmdState.cSTA_VPC_StabilizeBusy: 
        THIS^.sta_StabilizeVacuum();
	cSTA_RUNBusy: 
        THIS^.sta_RUNBusy();
    cSTA_RUN: 
        THIS^.sta_RUN();
END_CASE;
END_METHOD

END_FUNCTION_BLOCK

// POUs/Controller/Lvl3/BaseCtrlModule/FB_CtrlModule
FUNCTION_BLOCK FB_CtrlModule EXTENDS FB_CtrlBase
VAR_INPUT
	// Emergency circuit OK
	In_bolEmoOk: BOOL;
	// signals that next module is ready
	In_bolReady: BOOL;
END_VAR
VAR_OUTPUT
	// signals that this module is ready
	Out_bolReady: BOOL;
END_VAR
VAR
	/// Timeout supervision of Keep alive Toggle Bit
	udinTimeToggle_ms: UDINT;
	/// Specific interface struct
	SIf_MOD: T_Ctrl_SIf_MOD;
	uinGroupIndex: UINT;
	intCheckCounter: INT;
	uinMaxNrOfGroups: UINT := Base_Const.cMaxNrOfChilds;
	/// List of sequences
	aListOfSeq: ARRAY[0..Base_Const.cMaxNrOfChilds] OF T_Sequence;
	usiNumOfSeq: USINT := 0;
	usiNumOfValidPointerSeqChild: USINT := 0;
	/// [ms] List of waiting times for run sequence until the next group will execute
	/// If wait time is zero, next group will be directly executed after current group.  
	///	aListOfRunGrpWaitTime_ms: ARRAY[0..Base_Const.cMaxNrOfChilds] OF UDINT;
	usiNumOfRunGrpWaitTime: USINT := 0;
	/// [ms] List of waiting times for stop sequence until the next group will execute
	/// If wait time is zero, next group will be directly executed after current group. 
	///	aListOfStopGrpWaitTime_ms: ARRAY[0..Base_Const.cMaxNrOfChilds] OF UDINT;
	usiNumOfStopGrpWaitTime: USINT := 0;
	/// Array includes all registered childs of type IBuffer
	a_IBufferChildCtrl: ARRAY[0..Base_Const.cMaxNrOfChilds] OF IBuffer;
	a_IBufferFullChildCtrl: ARRAY[0..Base_Const.cMaxNrOfChilds] OF IBuffer;
	usiNumOfIBufferChild: USINT;
	usiNumOfIBufferFullChild: USINT;
	/// Counter
	ii: INT;
END_VAR
VAR CONSTANT
	/// sub States for run and stop sequences
	cSTA_SUB_INITIALIZED: INT := 500;
	cSTA_SUB_SEND_GROUP_CMD: INT := 502;
	cSTA_SUB_CHECK_GROUP_STATUS: INT := 504;
	cSTA_SUB_WAIT: INT := 506;
	cSTA_SUB_FINISHED: INT := 508;
END_VAR

(*__________________________________________________________________________________________________
¦	
¦	Vistaprint Schweiz GmbH
¦	CH - 8401 Winterthur
¦
¦	www.vistaprint.ch - info@vistaprint.ch
¦___________________________________________________________________________________________________

Function desription:
Basic module controller implementation. This Controller should be the base father controller for all modules in shirt stream. 
e.g. used for ICL, ICB, Loading ...

Controller handle following basic functions:
--------------------------------------------
- Monitoring of common signals from cabinet
- Keep alive bit to line control
- General child handling RUN_busy, STOP_busy sequences and error handling

History:
Version		Date			Author		Comment
---------------------------------------------------------------------------------------------------
0.00.1		06.11.2013		AVM/DSC		Start history
0.00.2		14.11.2013		AVM/MRU		Changes in some methods
0.00.3		29.11.2013		AVM/MRU		Changes in IoInBridge
0.00.4		04.12.2013		AVM/MRU		Changes in Always - EOFFBusy
0.00.5		04.12.2013		AVM/MRU		Changes in Always - EOFFBusy at GeneralError
0.00.6		04.12.2013		AVM/MRU		Changes in Always - EOFFBusy if not in sta_EOFF 
0.00.7		05.12.2013		AVM/DSC		General revision of behaviour in case of emergency off (state EOFF) and general error (state ERROR).
										New handling for module specific interface.
0.00.8		06.12.2013		AVM/MRU		Add TSTOP in checkChildAlmClass
0.00.9		09.12.2013		AVM/DSC		BugFix in sub state "cSTA_SUB_CHECK_GROUP_STATUS" from run and stop sequence. Insert new "bolChecked" flag
						 				to detect if the sequence has been processed correctly.
0.00.10		11.12.2013		AVM/MRU		Clear pending command to prevent automatic recovery in sta_STOPBusy
0.00.11		13.01.2014		AVM/MRU		Bugzilla ID 03: BufferFull added
0.00.12		20.01.2014		AVM/MRU		EMO, general error reworked; AddRunGrp, AddStopGrp removed
										Timeout run/stop group added 
0.00.13		22.01.2014		AVM/MRU		Alternativ status for run sequence added
0.00.14		08.02.2014		VP/RE		Added bolStopReleaseHangers to CUR.

___________________________________________________________________________________________________*)


IF (SIf_MOD.Cur<>0) AND (SIf_MOD.Cfg<>0) AND (SIf_MOD.Par<>0) AND (SIf_MOD.In<>0) THEN // cyclic call enabled
	SUPER^();
END_IF;

METHOD AddIBufferChilds
VAR_INPUT
	pFB_ChildTypeIBuffer: POINTER TO FB_IBuffer;
END_VAR
// Method add childs with type of IBuffer to the array
IF (usiNumOfIBufferChild <= (Base_Const.cMaxNrOfChilds-1)) THEN
	// Add child controller to list
	a_IBufferChildCtrl[usiNumOfIBufferChild] := pFB_ChildTypeIBuffer^;
	// Inc. number of IBuffer childs
	usiNumOfIBufferChild:= usiNumOfIBufferChild+1;
END_IF
END_METHOD

METHOD AddIBufferFullChilds
VAR_INPUT
	pFB_ChildTypeIBuffer: POINTER TO FB_IBuffer;
END_VAR
// Method add childs with BufferFull information to the array
IF (usiNumOfIBufferFullChild <= (Base_Const.cMaxNrOfChilds-1)) THEN
	// Add child controller to list
	a_IBufferFullChildCtrl[usiNumOfIBufferFullChild] := pFB_ChildTypeIBuffer^;

	// Inc. number of IBufferFull childs
	usiNumOfIBufferFullChild:= usiNumOfIBufferFullChild+1;
END_IF
END_METHOD

METHOD AddSeqChild
VAR_INPUT
	stSequence: T_Sequence;
END_VAR
// Method add a sequence to list
IF (usiNumOfSeq <= (Base_Const.cMaxNrOfChilds-1)) THEN
	aListOfSeq[usiNumOfSeq].pChild:= stSequence.pChild;
	aListOfSeq[usiNumOfSeq].uinGroupRun:= stSequence.uinGroupRun;
	aListOfSeq[usiNumOfSeq].uinGroupStop:= stSequence.uinGroupStop;
	aListOfSeq[usiNumOfSeq].intCmdSeqRun:= stSequence.intCmdSeqRun;
	aListOfSeq[usiNumOfSeq].intStatusSeqRun:= stSequence.intStatusSeqRun;
	aListOfSeq[usiNumOfSeq].intStatusSeqRun2:= stSequence.intStatusSeqRun2;
	aListOfSeq[usiNumOfSeq].intCmdSeqStop:= stSequence.intCmdSeqStop;
	aListOfSeq[usiNumOfSeq].intStatusSeqStop:= stSequence.intStatusSeqStop;
	// Inc. number of sequence
	usiNumOfSeq:= usiNumOfSeq+1;
	// Check if the pointer is valid
	IF (stSequence.pChild<>0) THEN
		usiNumOfValidPointerSeqChild:= usiNumOfValidPointerSeqChild+1;
	END_IF
END_IF
END_METHOD

METHOD PROTECTED Always : BOOL
SUPER^.Always();

